  MoveL 1279 to (-195.45, 422.54, -1.48) mm, rotated rx 180 ry 0 rz 13.5 deg; joints [-3.576, -31.782, 134.338, -181.987, 89.848, 89.481, 155.176]
  MoveL 1280 to (-195.21, 422.52, -1.48) mm, rotated rx -180 ry 0 rz 13.48 deg; joints [-3.576, -31.791, 134.342, -181.987, 89.843, 89.481, 155.202]
  MoveL 1281 to (-194.97, 422.52, -1.48) mm, rotated rx 180 ry 0 rz 13.45 deg; joints [-3.576, -31.8, 134.346, -181.987, 89.838, 89.481, 155.229]
  Set speed (38.1 mm/s)
  MoveL 1282 to (-194.97, 421.25, -1.48) mm, rotated rx 180 ry 0 rz 13.52 deg; joints [-3.576, -31.894, 134.387, -181.987, 89.785, 89.483, 155.164]
  MoveL 1283 to (-195.61, 421.25, -1.47) mm, rotated rx 180 ry 0 rz 13.59 deg; joints [-3.576, -31.872, 134.377, -181.987, 89.798, 89.482, 155.093]
  Set speed (25.4 mm/s)
  MoveL 1284 to (-195.61, 421.25, -3.84) mm, rotated rx -180 ry 0 rz 13.59 deg; joints [-3.707, -31.873, 134.372, -182.114, 89.79, 89.454, 155.093]
  MoveL 1285 to (-195.61, 421.89, -4.48) mm, rotated rx 180 ry 0 rz 13.55 deg; joints [-3.742, -31.826, 134.349, -182.149, 89.814, 89.446, 155.125]
  Set speed (38.1 mm/s)
  MoveL 1286 to (-194.97, 422.52, -4.48) mm, rotated rx 180 ry 0 rz 13.45 deg; joints [-3.742, -31.8, 134.338, -182.149, 89.829, 89.445, 155.229]
  Set speed (76.2 mm/s)
  MoveL 1287 to (213.41, 422.52, -4.48) mm, rotated rx -180 ry 0 rz -38.12 deg; joints [-4.097, -49.127, 150.45, -182.187, 60.817, 89.337, 179]
  MoveL 1288 to (213.89, 422.53, -4.48) mm, rotated rx 180 ry 0 rz -38.17 deg; joints [-4.098, -49.152, 150.476, -182.187, 60.765, 89.336, 179]
  MoveL 1289 to (214.13, 422.55, -4.47) mm, rotated rx -180 ry 0 rz -38.19 deg; joints [-4.098, -49.161, 150.488, -182.187, 60.743, 89.336, 179]
  MoveL 1290 to (214.37, 422.59, -4.48) mm, rotated rx 180 ry 0 rz -38.22 deg; joints [-4.099, -49.169, 150.501, -182.187, 60.725, 89.336, 179]
  MoveL 1291 to (214.61, 422.65, -4.48) mm, rotated rx -180 ry 0 rz -38.24 deg; joints [-4.099, -49.173, 150.512, -182.187, 60.709, 89.335, 179]
  MoveL 1292 to (214.85, 422.74, -4.48) mm, rotated rx -180 ry 0 rz -38.26 deg; joints [-4.1, -49.175, 150.524, -182.187, 60.698, 89.334, 179]
  MoveL 1293 to (215.09, 422.84, -4.48) mm, rotated rx -180 ry 0 rz -38.28 deg; joints [-4.1, -49.174, 150.536, -182.187, 60.69, 89.334, 179]
  MoveL 1294 to (215.34, 422.97, -4.48) mm, rotated rx -180 ry 0 rz -38.3 deg; joints [-4.101, -49.17, 150.547, -182.187, 60.687, 89.333, 179]
  MoveL 1295 to (215.58, 423.13, -4.48) mm, rotated rx -180 ry 0 rz -38.32 deg; joints [-4.101, -49.161, 150.557, -182.186, 60.688, 89.332, 179]
  MoveL 1296 to (215.82, 423.33, -4.48) mm, rotated rx -180 ry 0 rz -38.33 deg; joints [-4.102, -49.148, 150.568, -182.186, 60.696, 89.33, 179]
  MoveL 1297 to (215.96, 423.46, -4.48) mm, rotated rx -180 ry 0 rz -38.34 deg; joints [-4.102, -49.138, 150.573, -182.186, 60.705, 89.33, 179]
  MoveL 1298 to (216.09, 423.6, -4.48) mm, rotated rx 180 ry 0 rz -38.35 deg; joints [-4.102, -49.127, 150.578, -182.186, 60.715, 89.329, 179]
  MoveL 1299 to (216.2, 423.73, -4.48) mm, rotated rx 180 ry 0 rz -38.35 deg; joints [-4.103, -49.115, 150.582, -182.186, 60.726, 89.328, 179]
  MoveL 1300 to (216.3, 423.87, -4.47) mm, rotated rx -180 ry 0 rz -38.36 deg; joints [-4.103, -49.102, 150.586, -182.186, 60.739, 89.327, 179]
  MoveL 1301 to (216.39, 424.01, -4.48) mm, rotated rx -180 ry 0 rz -38.36 deg; joints [-4.103, -49.089, 150.589, -182.185, 60.753, 89.326, 179]
  MoveL 1302 to (216.47, 424.15, -4.48) mm, rotated rx -180 ry 0 rz -38.36 deg; joints [-4.104, -49.075, 150.592, -182.185, 60.768, 89.326, 179]
  MoveL 1303 to (216.6, 424.39, -4.48) mm, rotated rx -180 ry 0 rz -38.36 deg; joints [-4.104, -49.049, 150.595, -182.185, 60.797, 89.324, 179]
  MoveL 1304 to (216.69, 424.63, -4.48) mm, rotated rx -180 ry 0 rz -38.36 deg; joints [-4.104, -49.023, 150.597, -182.185, 60.828, 89.323, 179]
  MoveL 1305 to (216.77, 424.87, -4.48) mm, rotated rx 180 ry 0 rz -38.35 deg; joints [-4.105, -48.995, 150.598, -182.185, 60.862, 89.322, 179]
  MoveL 1306 to (216.82, 425.11, -4.48) mm, rotated rx -180 ry 0 rz -38.34 deg; joints [-4.105, -48.966, 150.597, -182.184, 60.898, 89.32, 179]
  MoveL 1307 to (216.86, 425.35, -4.48) mm, rotated rx -180 ry 0 rz -38.33 deg; joints [-4.105, -48.936, 150.596, -182.184, 60.936, 89.319, 179]
  MoveL 1308 to (216.88, 425.59, -4.48) mm, rotated rx -180 ry 0 rz -38.32 deg; joints [-4.105, -48.905, 150.594, -182.184, 60.976, 89.318, 179]
  MoveL 1309 to (216.88, 426.08, -4.48) mm, rotated rx 180 ry 0 rz -38.3 deg; joints [-4.106, -48.841, 150.587, -182.183, 61.06, 89.315, 179]
  MoveL 1310 to (216.88, 426.56, -4.48) mm, rotated rx -180 ry 0 rz -38.27 deg; joints [-4.106, -48.777, 150.58, -182.183, 61.143, 89.313, 179]
  MoveL 1311 to (216.86, 426.8, -4.47) mm, rotated rx 180 ry 0 rz -38.26 deg; joints [-4.106, -48.744, 150.576, -182.182, 61.187, 89.312, 179]
  MoveL 1312 to (216.82, 427.04, -4.48) mm, rotated rx -180 ry 0 rz -38.24 deg; joints [-4.107, -48.71, 150.571, -182.182, 61.232, 89.311, 179]
  MoveL 1313 to (216.76, 427.29, -4.47) mm, rotated rx 180 ry 0 rz -38.22 deg; joints [-4.107, -48.675, 150.564, -182.182, 61.28, 89.31, 179]
  MoveL 1314 to (216.68, 427.53, -4.48) mm, rotated rx -180 ry 0 rz -38.2 deg; joints [-4.107, -48.639, 150.557, -182.182, 61.33, 89.308, 179]
  MoveL 1315 to (216.58, 427.77, -4.48) mm, rotated rx -180 ry 0 rz -38.17 deg; joints [-4.107, -48.602, 150.548, -182.182, 61.382, 89.307, 179]
  MoveL 1316 to (216.46, 428.01, -4.48) mm, rotated rx -180 ry 0 rz -38.15 deg; joints [-4.107, -48.564, 150.538, -182.181, 61.437, 89.306, 179]
  MoveL 1317 to (216.3, 428.26, -4.47) mm, rotated rx 180 ry 0 rz -38.12 deg; joints [-4.107, -48.523, 150.526, -182.181, 61.496, 89.305, 179]
  MoveL 1318 to (216.2, 428.39, -4.47) mm, rotated rx 180 ry 0 rz -38.1 deg; joints [-4.107, -48.5, 150.519, -182.181, 61.529, 89.305, 179]
  MoveL 1319 to (216.09, 428.53, -4.48) mm, rotated rx -180 ry 0 rz -38.08 deg; joints [-4.107, -48.476, 150.511, -182.181, 61.564, 89.304, 179]
  MoveL 1320 to (215.96, 428.66, -4.47) mm, rotated rx 180 ry 0 rz -38.06 deg; joints [-4.106, -48.452, 150.502, -182.181, 61.601, 89.304, 179]
  MoveL 1321 to (215.82, 428.8, -4.48) mm, rotated rx -180 ry 0 rz -38.04 deg; joints [-4.106, -48.427, 150.492, -182.181, 61.639, 89.303, 179]
  MoveL 1322 to (215.58, 428.99, -4.47) mm, rotated rx 180 ry 0 rz -38 deg; joints [-4.106, -48.389, 150.477, -182.18, 61.697, 89.303, 179]
  MoveL 1323 to (215.34, 429.15, -4.48) mm, rotated rx -180 ry 0 rz -37.97 deg; joints [-4.106, -48.355, 150.461, -182.18, 61.75, 89.302, 179]
  MoveL 1324 to (215.09, 429.28, -4.48) mm, rotated rx -180 ry 0 rz -37.93 deg; joints [-4.105, -48.326, 150.447, -182.18, 61.797, 89.302, 179]
  MoveL 1325 to (214.85, 429.39, -4.48) mm, rotated rx -180 ry 0 rz -37.9 deg; joints [-4.105, -48.299, 150.432, -182.18, 61.841, 89.301, 179]
  MoveL 1326 to (214.61, 429.47, -4.48) mm, rotated rx 180 ry 0 rz -37.87 deg; joints [-4.105, -48.276, 150.418, -182.18, 61.88, 89.301, 179]
  MoveL 1327 to (214.37, 429.53, -4.47) mm, rotated rx 180 ry 0 rz -37.84 deg; joints [-4.104, -48.255, 150.404, -182.18, 61.916, 89.301, 179]
  MoveL 1328 to (214.13, 429.58, -4.48) mm, rotated rx -180 ry 0 rz -37.82 deg; joints [-4.104, -48.237, 150.39, -182.18, 61.948, 89.301, 179]
  MoveL 1329 to (213.89, 429.6, -4.48) mm, rotated rx -180 ry 0 rz -37.79 deg; joints [-4.104, -48.222, 150.377, -182.18, 61.977, 89.302, 179]
  MoveL 1330 to (213.41, 429.6, -4.47) mm, rotated rx 180 ry 0 rz -37.74 deg; joints [-4.103, -48.196, 150.351, -182.18, 62.029, 89.302, 179]
  MoveL 1331 to (-194.97, 429.6, -4.48) mm, rotated rx 180 ry 0 rz 13.09 deg; joints [-3.743, -31.276, 134.105, -182.15, 90.119, 89.434, 155.59]
  MoveL 1332 to (-195.21, 429.6, -4.48) mm, rotated rx 180 ry 0 rz 13.12 deg; joints [-3.743, -31.268, 134.101, -182.15, 90.124, 89.434, 155.563]
  MoveL 1333 to (-195.45, 429.58, -4.47) mm, rotated rx -180 ry 0 rz 13.14 deg; joints [-3.743, -31.261, 134.098, -182.15, 90.128, 89.434, 155.535]
  MoveL 1334 to (-195.69, 429.55, -4.47) mm, rotated rx 180 ry 0 rz 13.17 deg; joints [-3.743, -31.256, 134.096, -182.15, 90.131, 89.434, 155.507]
  MoveL 1335 to (-195.93, 429.49, -4.48) mm, rotated rx 180 ry 0 rz 13.2 deg; joints [-3.743, -31.252, 134.094, -182.15, 90.133, 89.434, 155.477]
  MoveL 1336 to (-196.18, 429.42, -4.48) mm, rotated rx 180 ry 0 rz 13.23 deg; joints [-3.743, -31.249, 134.093, -182.15, 90.134, 89.434, 155.447]
  MoveL 1337 to (-196.42, 429.32, -4.48) mm, rotated rx 180 ry 0 rz 13.26 deg; joints [-3.743, -31.248, 134.092, -182.15, 90.135, 89.434, 155.415]
  MoveL 1338 to (-196.6, 429.23, -4.48) mm, rotated rx -180 ry 0 rz 13.29 deg; joints [-3.743, -31.249, 134.092, -182.15, 90.134, 89.434, 155.391]
  MoveL 1339 to (-196.78, 429.13, -4.48) mm, rotated rx 180 ry 0 rz 13.31 deg; joints [-3.743, -31.25, 134.093, -182.15, 90.133, 89.434, 155.366]
  MoveL 1340 to (-196.95, 429.01, -4.48) mm, rotated rx 180 ry 0 rz 13.34 deg; joints [-3.743, -31.253, 134.094, -182.15, 90.132, 89.434, 155.34]
  MoveL 1341 to (-197.13, 428.87, -4.48) mm, rotated rx 180 ry 0 rz 13.37 deg; joints [-3.743, -31.257, 134.096, -182.15, 90.13, 89.434, 155.313]
  MoveL 1342 to (-197.37, 428.65, -4.48) mm, rotated rx 180 ry 0 rz 13.4 deg; joints [-3.743, -31.265, 134.1, -182.15, 90.125, 89.434, 155.277]
  MoveL 1343 to (-197.56, 428.44, -4.48) mm, rotated rx -180 ry 0 rz 13.43 deg; joints [-3.743, -31.274, 134.104, -182.15, 90.12, 89.434, 155.245]
  MoveL 1344 to (-197.72, 428.22, -4.48) mm, rotated rx 180 ry 0 rz 13.46 deg; joints [-3.742, -31.285, 134.109, -182.15, 90.114, 89.434, 155.217]
  MoveL 1345 to (-197.85, 428.01, -4.47) mm, rotated rx 180 ry 0 rz 13.49 deg; joints [-3.742, -31.296, 134.114, -182.15, 90.108, 89.435, 155.191]
  MoveL 1346 to (-197.98, 427.77, -4.48) mm, rotated rx 180 ry 0 rz 13.51 deg; joints [-3.742, -31.31, 134.12, -182.15, 90.101, 89.435, 155.165]
  MoveL 1347 to (-198.08, 427.53, -4.48) mm, rotated rx 180 ry 0 rz 13.54 deg; joints [-3.742, -31.324, 134.126, -182.15, 90.093, 89.435, 155.141]
  MoveL 1348 to (-198.16, 427.29, -4.48) mm, rotated rx 180 ry 0 rz 13.56 deg; joints [-3.742, -31.339, 134.133, -182.15, 90.085, 89.435, 155.12]
  MoveL 1349 to (-198.21, 427.04, -4.48) mm, rotated rx 180 ry 0 rz 13.58 deg; joints [-3.742, -31.355, 134.14, -182.149, 90.076, 89.436, 155.102]
  MoveL 1350 to (-198.25, 426.8, -4.48) mm, rotated rx 180 ry 0 rz 13.59 deg; joints [-3.742, -31.372, 134.148, -182.149, 90.067, 89.436, 155.085]
  MoveL 1351 to (-198.27, 426.56, -4.48) mm, rotated rx -180 ry 0 rz 13.61 deg; joints [-3.742, -31.389, 134.155, -182.149, 90.057, 89.437, 155.071]
  MoveL 1352 to (-198.27, 426.08, -4.48) mm, rotated rx -180 ry 0 rz 13.63 deg; joints [-3.742, -31.424, 134.171, -182.149, 90.038, 89.437, 155.045]
  MoveL 1353 to (-198.27, 425.59, -4.48) mm, rotated rx 180 ry 0 rz 13.66 deg; joints [-3.742, -31.46, 134.187, -182.149, 90.018, 89.438, 155.021]
  MoveL 1354 to (-198.25, 425.35, -4.48) mm, rotated rx -180 ry 0 rz 13.67 deg; joints [-3.742, -31.478, 134.195, -182.149, 90.008, 89.438, 155.01]
  MoveL 1355 to (-198.22, 425.11, -4.48) mm, rotated rx -180 ry 0 rz 13.68 deg; joints [-3.742, -31.497, 134.204, -182.149, 89.997, 89.439, 155.002]
  MoveL 1356 to (-198.16, 424.87, -4.48) mm, rotated rx 180 ry 0 rz 13.68 deg; joints [-3.742, -31.517, 134.213, -182.149, 89.986, 89.439, 154.995]
  MoveL 1357 to (-198.09, 424.63, -4.48) mm, rotated rx -180 ry 0 rz 13.69 deg; joints [-3.742, -31.538, 134.222, -182.149, 89.975, 89.44, 154.991]
  MoveL 1358 to (-197.99, 424.39, -4.48) mm, rotated rx 180 ry 0 rz 13.69 deg; joints [-3.742, -31.559, 134.231, -182.149, 89.963, 89.44, 154.989]
  MoveL 1359 to (-197.87, 424.15, -4.47) mm, rotated rx 180 ry 0 rz 13.69 deg; joints [-3.742, -31.581, 134.241, -182.149, 89.951, 89.441, 154.991]
  MoveL 1360 to (-197.73, 423.93, -4.48) mm, rotated rx -180 ry 0 rz 13.69 deg; joints [-3.742, -31.602, 134.25, -182.149, 89.939, 89.441, 154.994]
  MoveL 1361 to (-197.57, 423.71, -4.48) mm, rotated rx 180 ry 0 rz 13.68 deg; joints [-3.742, -31.623, 134.26, -182.149, 89.927, 89.441, 155.001]
  MoveL 1362 to (-197.38, 423.49, -4.48) mm, rotated rx 180 ry 0 rz 13.67 deg; joints [-3.742, -31.646, 134.27, -182.149, 89.914, 89.442, 155.011]
  MoveL 1363 to (-197.14, 423.27, -4.48) mm, rotated rx -180 ry 0 rz 13.65 deg; joints [-3.742, -31.671, 134.281, -182.149, 89.901, 89.442, 155.026]
  MoveL 1364 to (-196.96, 423.13, -4.47) mm, rotated rx 180 ry 0 rz 13.64 deg; joints [-3.742, -31.687, 134.288, -182.149, 89.892, 89.443, 155.038]
  MoveL 1365 to (-196.78, 423, -4.47) mm, rotated rx 180 ry 0 rz 13.63 deg; joints [-3.742, -31.703, 134.295, -182.149, 89.883, 89.443, 155.052]
  MoveL 1366 to (-196.6, 422.9, -4.47) mm, rotated rx 180 ry 0 rz 13.61 deg; joints [-3.742, -31.717, 134.301, -182.149, 89.875, 89.443, 155.067]
  MoveL 1367 to (-196.42, 422.81, -4.48) mm, rotated rx -180 ry 0 rz 13.6 deg; joints [-3.742, -31.73, 134.307, -182.149, 89.868, 89.444, 155.083]
  MoveL 1368 to (-196.18, 422.71, -4.48) mm, rotated rx -180 ry 0 rz 13.58 deg; joints [-3.742, -31.745, 134.314, -182.149, 89.859, 89.444, 155.104]
  MoveL 1369 to (-195.93, 422.63, -4.48) mm, rotated rx 180 ry 0 rz 13.55 deg; joints [-3.742, -31.759, 134.32, -182.149, 89.852, 89.444, 155.127]
  MoveL 1370 to (-195.69, 422.58, -4.47) mm, rotated rx 180 ry 0 rz 13.53 deg; joints [-3.742, -31.771, 134.325, -182.149, 89.845, 89.445, 155.151]
  MoveL 1371 to (-195.45, 422.54, -4.48) mm, rotated rx 180 ry 0 rz 13.5 deg; joints [-3.742, -31.782, 134.33, -182.149, 89.839, 89.445, 155.176]
  MoveL 1372 to (-195.21, 422.52, -4.48) mm, rotated rx 180 ry 0 rz 13.48 deg; joints [-3.742, -31.792, 134.335, -182.149, 89.833, 89.445, 155.202]
  MoveL 1373 to (-194.97, 422.52, -4.48) mm, rotated rx 180 ry 0 rz 13.45 deg; joints [-3.742, -31.8, 134.338, -182.149, 89.829, 89.445, 155.229]
  Set speed (38.1 mm/s)
  MoveL 1374 to (-194.97, 421.25, -4.48) mm, rotated rx -180 ry 0 rz 13.52 deg; joints [-3.742, -31.894, 134.38, -182.149, 89.776, 89.447, 155.164]
  MoveL 1375 to (-195.61, 421.25, -4.48) mm, rotated rx -180 ry 0 rz 13.59 deg; joints [-3.742, -31.873, 134.37, -182.149, 89.788, 89.447, 155.093]
  Set speed (25.4 mm/s)
  MoveL 1376 to (-195.61, 421.25, -6.84) mm, rotated rx 180 ry 0 rz 13.59 deg; joints [-3.872, -31.873, 134.364, -182.276, 89.78, 89.419, 155.093]
  MoveL 1377 to (-195.61, 421.89, -7.47) mm, rotated rx 180 ry 0 rz 13.55 deg; joints [-3.907, -31.826, 134.341, -182.311, 89.804, 89.41, 155.125]
  Set speed (38.1 mm/s)
  MoveL 1378 to (-194.97, 422.52, -7.48) mm, rotated rx 180 ry 0 rz 13.45 deg; joints [-3.907, -31.801, 134.33, -182.311, 89.818, 89.41, 155.229]
  Set speed (76.2 mm/s)
  MoveL 1379 to (213.41, 422.52, -7.47) mm, rotated rx 180 ry 0 rz -38.12 deg; joints [-4.291, -49.127, 150.441, -182.356, 60.805, 89.294, 179]
  MoveL 1380 to (213.89, 422.53, -7.48) mm, rotated rx -180 ry 0 rz -38.17 deg; joints [-4.291, -49.152, 150.466, -182.356, 60.754, 89.293, 179]
  MoveL 1381 to (214.13, 422.55, -7.48) mm, rotated rx -180 ry 0 rz -38.19 deg; joints [-4.292, -49.162, 150.479, -182.356, 60.732, 89.293, 179]
  MoveL 1382 to (214.37, 422.59, -7.48) mm, rotated rx 180 ry 0 rz -38.22 deg; joints [-4.292, -49.169, 150.491, -182.356, 60.713, 89.293, 179]
  MoveL 1383 to (214.61, 422.65, -7.48) mm, rotated rx -180 ry 0 rz -38.24 deg; joints [-4.293, -49.174, 150.503, -182.356, 60.698, 89.292, 179]
  MoveL 1384 to (214.85, 422.74, -7.47) mm, rotated rx 180 ry 0 rz -38.26 deg; joints [-4.293, -49.176, 150.515, -182.356, 60.686, 89.291, 179]
  MoveL 1385 to (215.09, 422.84, -7.47) mm, rotated rx 180 ry 0 rz -38.28 deg; joints [-4.294, -49.175, 150.526, -182.355, 60.678, 89.29, 179]
  MoveL 1386 to (215.34, 422.97, -7.48) mm, rotated rx -180 ry 0 rz -38.3 deg; joints [-4.294, -49.17, 150.537, -182.355, 60.675, 89.289, 179]
  MoveL 1387 to (215.58, 423.13, -7.48) mm, rotated rx -180 ry 0 rz -38.32 deg; joints [-4.295, -49.162, 150.548, -182.355, 60.677, 89.288, 179]
  MoveL 1388 to (215.82, 423.33, -7.47) mm, rotated rx 180 ry 0 rz -38.33 deg; joints [-4.296, -49.149, 150.558, -182.355, 60.685, 89.287, 179]
  MoveL 1389 to (215.96, 423.46, -7.48) mm, rotated rx -180 ry 0 rz -38.34 deg; joints [-4.296, -49.139, 150.564, -182.355, 60.693, 89.286, 179]
  MoveL 1390 to (216.09, 423.6, -7.48) mm, rotated rx -180 ry 0 rz -38.35 deg; joints [-4.296, -49.128, 150.569, -182.355, 60.703, 89.285, 179]
  MoveL 1391 to (216.2, 423.73, -7.48) mm, rotated rx 180 ry 0 rz -38.35 deg; joints [-4.297, -49.116, 150.573, -182.354, 60.714, 89.284, 179]
  MoveL 1392 to (216.3, 423.87, -7.48) mm, rotated rx -180 ry 0 rz -38.36 deg; joints [-4.297, -49.103, 150.577, -182.354, 60.727, 89.283, 179]
  MoveL 1393 to (216.39, 424.01, -7.48) mm, rotated rx 180 ry 0 rz -38.36 deg; joints [-4.297, -49.09, 150.58, -182.354, 60.741, 89.283, 179]
  MoveL 1394 to (216.47, 424.15, -7.48) mm, rotated rx -180 ry 0 rz -38.36 deg; joints [-4.298, -49.076, 150.582, -182.354, 60.756, 89.282, 179]
  MoveL 1395 to (216.6, 424.39, -7.48) mm, rotated rx -180 ry 0 rz -38.36 deg; joints [-4.298, -49.05, 150.585, -182.354, 60.785, 89.28, 179]
  MoveL 1396 to (216.69, 424.63, -7.48) mm, rotated rx 180 ry 0 rz -38.36 deg; joints [-4.298, -49.024, 150.587, -182.353, 60.817, 89.279, 179]
  MoveL 1397 to (216.77, 424.87, -7.47) mm, rotated rx -180 ry 0 rz -38.35 deg; joints [-4.299, -48.996, 150.588, -182.353, 60.85, 89.277, 179]
  MoveL 1398 to (216.82, 425.11, -7.47) mm, rotated rx -180 ry 0 rz -38.34 deg; joints [-4.299, -48.967, 150.588, -182.353, 60.886, 89.276, 179]
  MoveL 1399 to (216.86, 425.35, -7.48) mm, rotated rx -180 ry 0 rz -38.33 deg; joints [-4.299, -48.937, 150.587, -182.353, 60.924, 89.275, 179]
  MoveL 1400 to (216.88, 425.59, -7.47) mm, rotated rx 180 ry 0 rz -38.32 deg; joints [-4.3, -48.906, 150.584, -182.352, 60.964, 89.273, 179]
  MoveL 1401 to (216.88, 426.08, -7.48) mm, rotated rx -180 ry 0 rz -38.3 deg; joints [-4.3, -48.842, 150.578, -182.352, 61.048, 89.271, 179]
  MoveL 1402 to (216.88, 427.04, -7.47) mm, rotated rx 180 ry 0 rz -38.24 deg; joints [-4.301, -48.714, 150.564, -182.351, 61.214, 89.266, 179]
  MoveL 1403 to (216.86, 427.29, -7.48) mm, rotated rx -180 ry 0 rz -38.23 deg; joints [-4.301, -48.682, 150.56, -182.35, 61.257, 89.264, 179]
  MoveL 1404 to (216.83, 427.53, -7.48) mm, rotated rx -180 ry 0 rz -38.21 deg; joints [-4.301, -48.648, 150.555, -182.35, 61.302, 89.263, 179]
  MoveL 1405 to (216.78, 427.77, -7.48) mm, rotated rx -180 ry 0 rz -38.19 deg; joints [-4.301, -48.614, 150.549, -182.35, 61.349, 89.262, 179]
  MoveL 1406 to (216.71, 428.01, -7.47) mm, rotated rx 180 ry 0 rz -38.17 deg; joints [-4.301, -48.578, 150.542, -182.35, 61.398, 89.261, 179]
  MoveL 1407 to (216.63, 428.21, -7.48) mm, rotated rx -180 ry 0 rz -38.16 deg; joints [-4.301, -48.548, 150.535, -182.349, 61.441, 89.26, 179]
  MoveL 1408 to (216.54, 428.41, -7.48) mm, rotated rx 180 ry 0 rz -38.13 deg; joints [-4.301, -48.517, 150.527, -182.349, 61.484, 89.259, 179]
  MoveL 1409 to (216.43, 428.61, -7.48) mm, rotated rx 180 ry 0 rz -38.11 deg; joints [-4.301, -48.485, 150.518, -182.349, 61.53, 89.258, 179]
  MoveL 1410 to (216.3, 428.81, -7.48) mm, rotated rx -180 ry 0 rz -38.09 deg; joints [-4.301, -48.452, 150.509, -182.349, 61.578, 89.257, 179]
  MoveL 1411 to (216.16, 428.99, -7.48) mm, rotated rx -180 ry 0 rz -38.06 deg; joints [-4.301, -48.42, 150.498, -182.348, 61.624, 89.256, 179]
  MoveL 1412 to (215.99, 429.18, -7.48) mm, rotated rx -180 ry 0 rz -38.04 deg; joints [-4.301, -48.387, 150.487, -182.348, 61.673, 89.255, 179]
  MoveL 1413 to (215.78, 429.38, -7.48) mm, rotated rx -180 ry 0 rz -38 deg; joints [-4.301, -48.35, 150.473, -182.348, 61.729, 89.255, 179]
  MoveL 1414 to (215.57, 429.55, -7.48) mm, rotated rx -180 ry 0 rz -37.97 deg; joints [-4.301, -48.317, 150.459, -182.348, 61.78, 89.254, 179]
  MoveL 1415 to (215.39, 429.67, -7.48) mm, rotated rx -180 ry 0 rz -37.94 deg; joints [-4.3, -48.291, 150.447, -182.348, 61.82, 89.254, 179]
  MoveL 1416 to (215.21, 429.78, -7.48) mm, rotated rx -180 ry 0 rz -37.92 deg; joints [-4.3, -48.268, 150.436, -182.348, 61.857, 89.253, 179]
  MoveL 1417 to (215.02, 429.87, -7.47) mm, rotated rx 180 ry 0 rz -37.9 deg; joints [-4.3, -48.246, 150.425, -182.348, 61.892, 89.253, 179]
  MoveL 1418 to (214.84, 429.94, -7.48) mm, rotated rx -180 ry 0 rz -37.87 deg; joints [-4.3, -48.227, 150.414, -182.348, 61.924, 89.253, 179]
  MoveL 1419 to (214.61, 430.02, -7.48) mm, rotated rx 180 ry 0 rz -37.84 deg; joints [-4.299, -48.204, 150.4, -182.347, 61.962, 89.253, 179]
  MoveL 1420 to (214.37, 430.08, -7.47) mm, rotated rx 180 ry 0 rz -37.81 deg; joints [-4.299, -48.184, 150.387, -182.347, 61.997, 89.253, 179]
  MoveL 1421 to (214.13, 430.13, -7.47) mm, rotated rx 180 ry 0 rz -37.79 deg; joints [-4.298, -48.166, 150.373, -182.347, 62.029, 89.253, 179]
  MoveL 1422 to (213.89, 430.15, -7.48) mm, rotated rx -180 ry 0 rz -37.76 deg; joints [-4.298, -48.151, 150.36, -182.347, 62.058, 89.253, 179]
  MoveL 1423 to (213.41, 430.15, -7.48) mm, rotated rx -180 ry 0 rz -37.71 deg; joints [-4.297, -48.125, 150.334, -182.347, 62.11, 89.254, 179]
  MoveL 1424 to (-194.49, 430.15, -7.48) mm, rotated rx -180 ry 0 rz 13.01 deg; joints [-3.908, -31.252, 134.086, -182.311, 90.123, 89.397, 155.671]
  MoveL 1425 to (-195.36, 430.14, -7.48) mm, rotated rx -180 ry 0 rz 13.11 deg; joints [-3.908, -31.223, 134.073, -182.311, 90.138, 89.397, 155.573]
  MoveL 1426 to (-195.58, 430.12, -7.48) mm, rotated rx 180 ry 0 rz 13.13 deg; joints [-3.908, -31.218, 134.07, -182.311, 90.141, 89.396, 155.548]
  MoveL 1427 to (-195.8, 430.08, -7.48) mm, rotated rx 180 ry 0 rz 13.16 deg; joints [-3.908, -31.214, 134.068, -182.311, 90.144, 89.396, 155.522]
  MoveL 1428 to (-196.02, 430.02, -7.47) mm, rotated rx 180 ry 0 rz 13.18 deg; joints [-3.908, -31.211, 134.067, -182.311, 90.146, 89.396, 155.495]
  MoveL 1429 to (-196.24, 429.94, -7.47) mm, rotated rx 180 ry 0 rz 13.21 deg; joints [-3.908, -31.209, 134.066, -182.311, 90.147, 89.396, 155.467]
  MoveL 1430 to (-196.42, 429.87, -7.48) mm, rotated rx 180 ry 0 rz 13.24 deg; joints [-3.908, -31.208, 134.066, -182.311, 90.147, 89.396, 155.443]
  MoveL 1431 to (-196.56, 429.79, -7.48) mm, rotated rx 180 ry 0 rz 13.26 deg; joints [-3.908, -31.209, 134.066, -182.311, 90.147, 89.396, 155.423]
  MoveL 1432 to (-196.71, 429.71, -7.48) mm, rotated rx 180 ry 0 rz 13.28 deg; joints [-3.908, -31.21, 134.067, -182.311, 90.146, 89.396, 155.403]
  MoveL 1433 to (-196.86, 429.62, -7.48) mm, rotated rx 180 ry 0 rz 13.3 deg; joints [-3.908, -31.212, 134.068, -182.311, 90.145, 89.396, 155.382]
  MoveL 1434 to (-197.01, 429.52, -7.48) mm, rotated rx 180 ry 0 rz 13.32 deg; joints [-3.908, -31.214, 134.069, -182.311, 90.144, 89.396, 155.36]
  MoveL 1435 to (-197.15, 429.4, -7.48) mm, rotated rx 180 ry 0 rz 13.34 deg; joints [-3.908, -31.218, 134.07, -182.311, 90.141, 89.396, 155.338]
  MoveL 1436 to (-197.3, 429.27, -7.48) mm, rotated rx 180 ry 0 rz 13.36 deg; joints [-3.908, -31.223, 134.073, -182.311, 90.139, 89.396, 155.315]
  MoveL 1437 to (-197.46, 429.1, -7.48) mm, rotated rx 180 ry 0 rz 13.39 deg; joints [-3.908, -31.23, 134.076, -182.311, 90.135, 89.397, 155.29]
  MoveL 1438 to (-197.6, 428.94, -7.48) mm, rotated rx 180 ry 0 rz 13.41 deg; joints [-3.908, -31.237, 134.079, -182.311, 90.131, 89.397, 155.266]
  MoveL 1439 to (-197.76, 428.71, -7.48) mm, rotated rx 180 ry 0 rz 13.44 deg; joints [-3.908, -31.248, 134.084, -182.311, 90.125, 89.397, 155.236]
  MoveL 1440 to (-197.9, 428.47, -7.48) mm, rotated rx 180 ry 0 rz 13.47 deg; joints [-3.908, -31.261, 134.09, -182.311, 90.118, 89.397, 155.209]
  MoveL 1441 to (-198.01, 428.24, -7.47) mm, rotated rx -180 ry 0 rz 13.49 deg; joints [-3.908, -31.274, 134.096, -182.311, 90.111, 89.398, 155.185]
  MoveL 1442 to (-198.1, 428.01, -7.48) mm, rotated rx 180 ry 0 rz 13.52 deg; joints [-3.908, -31.288, 134.102, -182.311, 90.103, 89.398, 155.163]
  MoveL 1443 to (-198.17, 427.77, -7.47) mm, rotated rx -180 ry 0 rz 13.54 deg; joints [-3.908, -31.304, 134.109, -182.311, 90.094, 89.398, 155.143]
  MoveL 1444 to (-198.23, 427.53, -7.47) mm, rotated rx -180 ry 0 rz 13.55 deg; joints [-3.908, -31.32, 134.116, -182.311, 90.086, 89.399, 155.125]
  MoveL 1445 to (-198.26, 427.29, -7.48) mm, rotated rx -180 ry 0 rz 13.57 deg; joints [-3.908, -31.336, 134.124, -182.311, 90.076, 89.399, 155.109]
  MoveL 1446 to (-198.27, 427.04, -7.48) mm, rotated rx 180 ry 0 rz 13.58 deg; joints [-3.908, -31.354, 134.131, -182.311, 90.067, 89.399, 155.095]
  MoveL 1447 to (-198.27, 426.08, -7.48) mm, rotated rx -180 ry 0 rz 13.63 deg; joints [-3.908, -31.425, 134.163, -182.311, 90.027, 89.401, 155.045]
  MoveL 1448 to (-198.27, 425.59, -7.48) mm, rotated rx 180 ry 0 rz 13.66 deg; joints [-3.908, -31.461, 134.179, -182.311, 90.008, 89.402, 155.021]
  MoveL 1449 to (-198.25, 425.35, -7.48) mm, rotated rx -180 ry 0 rz 13.67 deg; joints [-3.908, -31.479, 134.187, -182.311, 89.997, 89.402, 155.01]
  MoveL 1450 to (-198.22, 425.11, -7.48) mm, rotated rx 180 ry 0 rz 13.68 deg; joints [-3.908, -31.498, 134.196, -182.311, 89.987, 89.403, 155.002]
  MoveL 1451 to (-198.16, 424.87, -7.47) mm, rotated rx 180 ry 0 rz 13.68 deg; joints [-3.908, -31.518, 134.205, -182.311, 89.976, 89.403, 154.995]
  MoveL 1452 to (-198.09, 424.63, -7.48) mm, rotated rx -180 ry 0 rz 13.69 deg; joints [-3.908, -31.538, 134.214, -182.311, 89.965, 89.404, 154.991]
  MoveL 1453 to (-197.99, 424.39, -7.48) mm, rotated rx -180 ry 0 rz 13.69 deg; joints [-3.908, -31.56, 134.223, -182.311, 89.953, 89.404, 154.989]
  MoveL 1454 to (-197.87, 424.15, -7.47) mm, rotated rx 180 ry 0 rz 13.69 deg; joints [-3.908, -31.582, 134.233, -182.311, 89.941, 89.405, 154.991]
  MoveL 1455 to (-197.73, 423.93, -7.47) mm, rotated rx 180 ry 0 rz 13.69 deg; joints [-3.908, -31.602, 134.242, -182.311, 89.929, 89.405, 154.994]
  MoveL 1456 to (-197.57, 423.71, -7.47) mm, rotated rx 180 ry 0 rz 13.68 deg; joints [-3.908, -31.624, 134.252, -182.311, 89.917, 89.406, 155.001]
  MoveL 1457 to (-197.38, 423.49, -7.48) mm, rotated rx -180 ry 0 rz 13.67 deg; joints [-3.908, -31.647, 134.262, -182.311, 89.904, 89.406, 155.011]
  MoveL 1458 to (-197.14, 423.27, -7.47) mm, rotated rx 180 ry 0 rz 13.65 deg; joints [-3.908, -31.671, 134.273, -182.311, 89.891, 89.407, 155.026]
  MoveL 1459 to (-196.96, 423.13, -7.48) mm, rotated rx -180 ry 0 rz 13.64 deg; joints [-3.908, -31.688, 134.28, -182.311, 89.881, 89.407, 155.038]
  MoveL 1460 to (-196.78, 423, -7.47) mm, rotated rx 180 ry 0 rz 13.63 deg; joints [-3.908, -31.703, 134.287, -182.311, 89.873, 89.407, 155.052]
  MoveL 1461 to (-196.6, 422.9, -7.47) mm, rotated rx 180 ry 0 rz 13.61 deg; joints [-3.908, -31.717, 134.293, -182.311, 89.865, 89.408, 155.067]
  MoveL 1462 to (-196.42, 422.81, -7.48) mm, rotated rx 180 ry 0 rz 13.6 deg; joints [-3.908, -31.73, 134.299, -182.311, 89.858, 89.408, 155.083]
  MoveL 1463 to (-196.18, 422.71, -7.48) mm, rotated rx -180 ry 0 rz 13.58 deg; joints [-3.908, -31.746, 134.306, -182.311, 89.849, 89.408, 155.104]
  MoveL 1464 to (-195.93, 422.63, -7.48) mm, rotated rx -180 ry 0 rz 13.55 deg; joints [-3.908, -31.76, 134.312, -182.311, 89.842, 89.409, 155.127]
  MoveL 1465 to (-195.69, 422.58, -7.48) mm, rotated rx -180 ry 0 rz 13.53 deg; joints [-3.908, -31.772, 134.317, -182.311, 89.835, 89.409, 155.151]
  MoveL 1466 to (-195.45, 422.54, -7.48) mm, rotated rx 180 ry 0 rz 13.5 deg; joints [-3.908, -31.783, 134.322, -182.311, 89.829, 89.409, 155.176]
  MoveL 1467 to (-195.21, 422.52, -7.47) mm, rotated rx -180 ry 0 rz 13.48 deg; joints [-3.908, -31.793, 134.327, -182.311, 89.823, 89.409, 155.202]
  MoveL 1468 to (-194.97, 422.52, -7.48) mm, rotated rx 180 ry 0 rz 13.45 deg; joints [-3.907, -31.801, 134.33, -182.311, 89.818, 89.41, 155.229]
  Set speed (38.1 mm/s)
  MoveL 1469 to (-194.97, 421.25, -7.48) mm, rotated rx -180 ry 0 rz 13.52 deg; joints [-3.907, -31.895, 134.372, -182.31, 89.766, 89.412, 155.164]
  MoveL 1470 to (-195.61, 421.25, -7.47) mm, rotated rx 180 ry 0 rz 13.59 deg; joints [-3.907, -31.873, 134.362, -182.31, 89.778, 89.411, 155.093]
  Set speed (25.4 mm/s)
  MoveL 1471 to (-195.61, 421.25, -9.84) mm, rotated rx 180 ry 0 rz 13.59 deg; joints [-4.038, -31.874, 134.355, -182.438, 89.77, 89.383, 155.093]
  MoveL 1472 to (-195.61, 421.89, -10.48) mm, rotated rx -180 ry 0 rz 13.55 deg; joints [-4.073, -31.827, 134.333, -182.472, 89.794, 89.375, 155.125]
  Set speed (38.1 mm/s)
  MoveL 1473 to (-194.97, 422.52, -10.48) mm, rotated rx 180 ry 0 rz 13.45 deg; joints [-4.073, -31.802, 134.322, -182.472, 89.808, 89.374, 155.229]
  Set speed (76.2 mm/s)
  MoveL 1474 to (213.41, 422.52, -10.48) mm, rotated rx -180 ry 0 rz -38.12 deg; joints [-4.484, -49.128, 150.431, -182.524, 60.792, 89.251, 179]
  MoveL 1475 to (213.89, 422.53, -10.48) mm, rotated rx -180 ry 0 rz -38.17 deg; joints [-4.485, -49.153, 150.456, -182.524, 60.741, 89.251, 179]
  MoveL 1476 to (214.13, 422.55, -10.48) mm, rotated rx 180 ry 0 rz -38.19 deg; joints [-4.485, -49.163, 150.469, -182.524, 60.719, 89.25, 179]
  MoveL 1477 to (214.37, 422.59, -10.47) mm, rotated rx 180 ry 0 rz -38.22 deg; joints [-4.486, -49.17, 150.481, -182.524, 60.7, 89.25, 179]
  MoveL 1478 to (214.61, 422.65, -10.48) mm, rotated rx -180 ry 0 rz -38.24 deg; joints [-4.486, -49.175, 150.493, -182.524, 60.685, 89.249, 179]
  MoveL 1479 to (214.85, 422.74, -10.48) mm, rotated rx -180 ry 0 rz -38.26 deg; joints [-4.487, -49.177, 150.505, -182.524, 60.673, 89.248, 179]
  MoveL 1480 to (215.09, 422.84, -10.48) mm, rotated rx 180 ry 0 rz -38.28 deg; joints [-4.488, -49.176, 150.516, -182.524, 60.666, 89.247, 179]
  MoveL 1481 to (215.34, 422.97, -10.48) mm, rotated rx -180 ry 0 rz -38.3 deg; joints [-4.488, -49.171, 150.527, -182.524, 60.662, 89.246, 179]
  MoveL 1482 to (215.58, 423.13, -10.48) mm, rotated rx 180 ry 0 rz -38.32 deg; joints [-4.489, -49.163, 150.538, -182.524, 60.664, 89.245, 179]
  MoveL 1483 to (215.82, 423.33, -10.48) mm, rotated rx -180 ry 0 rz -38.33 deg; joints [-4.489, -49.15, 150.548, -182.524, 60.672, 89.244, 179]
  MoveL 1484 to (215.96, 423.46, -10.48) mm, rotated rx -180 ry 0 rz -38.34 deg; joints [-4.49, -49.14, 150.554, -182.523, 60.68, 89.243, 179]
  MoveL 1485 to (216.09, 423.6, -10.48) mm, rotated rx 180 ry 0 rz -38.35 deg; joints [-4.49, -49.128, 150.559, -182.523, 60.69, 89.242, 179]
  MoveL 1486 to (216.2, 423.73, -10.48) mm, rotated rx -180 ry 0 rz -38.35 deg; joints [-4.491, -49.117, 150.563, -182.523, 60.702, 89.241, 179]
  MoveL 1487 to (216.3, 423.87, -10.48) mm, rotated rx -180 ry 0 rz -38.36 deg; joints [-4.491, -49.104, 150.566, -182.523, 60.714, 89.24, 179]
  MoveL 1488 to (216.39, 424.01, -10.47) mm, rotated rx 180 ry 0 rz -38.36 deg; joints [-4.491, -49.091, 150.569, -182.523, 60.728, 89.239, 179]
  MoveL 1489 to (216.47, 424.15, -10.48) mm, rotated rx -180 ry 0 rz -38.36 deg; joints [-4.491, -49.077, 150.572, -182.523, 60.744, 89.238, 179]
  MoveL 1490 to (216.69, 424.27, -10.47) mm, rotated rx 180 ry 0 rz -38.38 deg; joints [-4.492, -49.072, 150.582, -182.522, 60.741, 89.237, 179]
  MoveL 1491 to (219.83, 424.27, -10.48) mm, rotated rx -180 ry 0 rz -38.71 deg; joints [-4.498, -49.236, 150.748, -182.523, 60.408, 89.233, 179]
  MoveL 1492 to (220.05, 424.15, -10.47) mm, rotated rx 180 ry 0 rz -38.74 deg; joints [-4.498, -49.264, 150.761, -182.523, 60.363, 89.233, 179]
  MoveL 1493 to (220.05, 53.41, -10.47) mm, rotated rx -180 ry 0 rz -47.68 deg; joints [-4.3, -87.184, 146.455, -190.693, 9.341, 98.376, 179]
  MoveL 1494 to (219.83, 53.17, -10.47) mm, rotated rx 180 ry 0 rz -47.72 deg; joints [-4.299, -87.185, 146.415, -190.774, 9.257, 98.458, 179]
  MoveL 1495 to (-199.12, 53.17, -10.47) mm, rotated rx 180 ry 0 rz 63.73 deg; joints [-4.039, -53.792, 140.61, -182.536, 74.12, 90.068, 104.952]
  MoveL 1496 to (-199.7, 53.18, -10.48) mm, rotated rx -180 ry 0 rz 63.77 deg; joints [-4.039, -53.744, 140.603, -182.536, 74.162, 90.066, 104.91]
  MoveL 1497 to (-199.9, 53.41, -10.48) mm, rotated rx -180 ry 0 rz 63.72 deg; joints [-4.039, -53.723, 140.6, -182.535, 74.18, 90.065, 104.959]
  MoveL 1498 to (-199.9, 424.15, -10.48) mm, rotated rx 180 ry 0 rz 13.91 deg; joints [-4.074, -31.512, 134.193, -182.473, 89.969, 89.367, 154.766]
  MoveL 1499 to (-199.7, 424.27, -10.48) mm, rotated rx 180 ry 0 rz 13.89 deg; joints [-4.074, -31.51, 134.192, -182.473, 89.97, 89.367, 154.794]
  MoveL 1500 to (-198.11, 424.27, -10.48) mm, rotated rx -180 ry 0 rz 13.71 deg; joints [-4.074, -31.565, 134.217, -182.473, 89.939, 89.368, 154.97]
  MoveL 1501 to (-197.87, 424.15, -10.48) mm, rotated rx 180 ry 0 rz 13.69 deg; joints [-4.074, -31.582, 134.225, -182.473, 89.93, 89.369, 154.991]
  MoveL 1502 to (-197.73, 423.93, -10.48) mm, rotated rx -180 ry 0 rz 13.69 deg; joints [-4.074, -31.603, 134.234, -182.473, 89.918, 89.369, 154.994]
  MoveL 1503 to (-197.57, 423.71, -10.48) mm, rotated rx 180 ry 0 rz 13.68 deg; joints [-4.074, -31.625, 134.243, -182.473, 89.906, 89.37, 155.001]
  MoveL 1504 to (-197.38, 423.49, -10.48) mm, rotated rx 180 ry 0 rz 13.67 deg; joints [-4.073, -31.648, 134.254, -182.472, 89.893, 89.37, 155.011]
  MoveL 1505 to (-197.14, 423.27, -10.48) mm, rotated rx 180 ry 0 rz 13.65 deg; joints [-4.073, -31.672, 134.264, -182.472, 89.88, 89.371, 155.026]
  MoveL 1506 to (-196.96, 423.13, -10.48) mm, rotated rx -180 ry 0 rz 13.64 deg; joints [-4.073, -31.689, 134.272, -182.472, 89.871, 89.371, 155.038]
  MoveL 1507 to (-196.78, 423, -10.48) mm, rotated rx 180 ry 0 rz 13.63 deg; joints [-4.073, -31.704, 134.279, -182.472, 89.862, 89.372, 155.052]
  MoveL 1508 to (-196.6, 422.9, -10.48) mm, rotated rx 180 ry 0 rz 13.61 deg; joints [-4.073, -31.718, 134.285, -182.472, 89.854, 89.372, 155.067]
  MoveL 1509 to (-196.42, 422.81, -10.47) mm, rotated rx -180 ry 0 rz 13.6 deg; joints [-4.073, -31.731, 134.29, -182.472, 89.847, 89.372, 155.083]
  MoveL 1510 to (-196.18, 422.71, -10.48) mm, rotated rx -180 ry 0 rz 13.58 deg; joints [-4.073, -31.747, 134.297, -182.472, 89.838, 89.373, 155.104]
  MoveL 1511 to (-195.93, 422.63, -10.48) mm, rotated rx -180 ry 0 rz 13.55 deg; joints [-4.073, -31.761, 134.303, -182.472, 89.831, 89.373, 155.127]
  MoveL 1512 to (-195.69, 422.58, -10.48) mm, rotated rx -180 ry 0 rz 13.53 deg; joints [-4.073, -31.773, 134.309, -182.472, 89.824, 89.373, 155.151]
  MoveL 1513 to (-195.45, 422.54, -10.48) mm, rotated rx 180 ry 0 rz 13.5 deg; joints [-4.073, -31.784, 134.314, -182.472, 89.818, 89.374, 155.176]
  MoveL 1514 to (-195.21, 422.52, -10.48) mm, rotated rx 180 ry 0 rz 13.48 deg; joints [-4.073, -31.794, 134.318, -182.472, 89.812, 89.374, 155.202]
  MoveL 1515 to (-194.97, 422.52, -10.48) mm, rotated rx 180 ry 0 rz 13.45 deg; joints [-4.073, -31.802, 134.322, -182.472, 89.808, 89.374, 155.229]
  Set speed (38.1 mm/s)
  MoveL 1516 to (-194.97, 421.25, -10.48) mm, rotated rx 180 ry 0 rz 13.52 deg; joints [-4.073, -31.896, 134.363, -182.472, 89.755, 89.376, 155.164]
  MoveL 1517 to (-195.61, 421.25, -10.48) mm, rotated rx 180 ry 0 rz 13.59 deg; joints [-4.073, -31.874, 134.354, -182.472, 89.767, 89.376, 155.093]
  Set speed (25.4 mm/s)
  MoveL 1518 to (-195.61, 421.25, -12.84) mm, rotated rx 180 ry 0 rz 13.59 deg; joints [-4.204, -31.875, 134.346, -182.6, 89.758, 89.348, 155.093]
  MoveL 1519 to (-195.61, 421.89, -13.47) mm, rotated rx 180 ry 0 rz 13.55 deg; joints [-4.239, -31.828, 134.324, -182.634, 89.782, 89.339, 155.125]
  Set speed (38.1 mm/s)
  MoveL 1520 to (-194.97, 422.52, -13.48) mm, rotated rx 180 ry 0 rz 13.45 deg; joints [-4.239, -31.803, 134.313, -182.634, 89.796, 89.339, 155.229]
  Set speed (76.2 mm/s)
  MoveL 1521 to (213.41, 422.52, -13.48) mm, rotated rx -180 ry 0 rz -38.12 deg; joints [-4.677, -49.129, 150.42, -182.693, 60.779, 89.208, 179]
  MoveL 1522 to (213.89, 422.53, -13.47) mm, rotated rx -180 ry 0 rz -38.17 deg; joints [-4.678, -49.154, 150.445, -182.693, 60.728, 89.208, 179]
  MoveL 1523 to (214.13, 422.55, -13.48) mm, rotated rx -180 ry 0 rz -38.19 deg; joints [-4.679, -49.164, 150.458, -182.693, 60.706, 89.207, 179]
  MoveL 1524 to (214.37, 422.59, -13.48) mm, rotated rx -180 ry 0 rz -38.22 deg; joints [-4.679, -49.171, 150.47, -182.693, 60.687, 89.207, 179]
  MoveL 1525 to (214.61, 422.65, -13.48) mm, rotated rx -180 ry 0 rz -38.24 deg; joints [-4.68, -49.176, 150.482, -182.693, 60.672, 89.206, 179]
  MoveL 1526 to (214.85, 422.74, -13.48) mm, rotated rx -180 ry 0 rz -38.26 deg; joints [-4.681, -49.178, 150.494, -182.693, 60.66, 89.205, 179]
  MoveL 1527 to (215.09, 422.84, -13.48) mm, rotated rx -180 ry 0 rz -38.28 deg; joints [-4.681, -49.176, 150.505, -182.693, 60.652, 89.204, 179]
  MoveL 1528 to (215.34, 422.97, -13.48) mm, rotated rx -180 ry 0 rz -38.3 deg; joints [-4.682, -49.172, 150.516, -182.693, 60.649, 89.203, 179]
  MoveL 1529 to (215.58, 423.13, -13.47) mm, rotated rx 180 ry 0 rz -38.32 deg; joints [-4.682, -49.164, 150.527, -182.693, 60.651, 89.202, 179]
  MoveL 1530 to (215.82, 423.33, -13.47) mm, rotated rx 180 ry 0 rz -38.33 deg; joints [-4.683, -49.151, 150.537, -182.692, 60.659, 89.2, 179]
  MoveL 1531 to (215.96, 423.46, -13.48) mm, rotated rx -180 ry 0 rz -38.34 deg; joints [-4.684, -49.14, 150.543, -182.692, 60.667, 89.199, 179]
  MoveL 1532 to (216.09, 423.6, -13.47) mm, rotated rx -180 ry 0 rz -38.35 deg; joints [-4.684, -49.129, 150.548, -182.692, 60.677, 89.198, 179]
  MoveL 1533 to (216.2, 423.73, -13.48) mm, rotated rx -180 ry 0 rz -38.35 deg; joints [-4.684, -49.117, 150.552, -182.692, 60.688, 89.197, 179]
  MoveL 1534 to (216.3, 423.87, -13.48) mm, rotated rx -180 ry 0 rz -38.36 deg; joints [-4.685, -49.105, 150.556, -182.692, 60.701, 89.196, 179]
  MoveL 1535 to (216.39, 424.01, -13.48) mm, rotated rx -180 ry 0 rz -38.36 deg; joints [-4.685, -49.091, 150.559, -182.691, 60.715, 89.195, 179]
  MoveL 1536 to (216.47, 424.15, -13.47) mm, rotated rx 180 ry 0 rz -38.36 deg; joints [-4.685, -49.077, 150.561, -182.691, 60.73, 89.194, 179]
  MoveL 1537 to (216.69, 424.27, -13.48) mm, rotated rx -180 ry 0 rz -38.38 deg; joints [-4.686, -49.073, 150.571, -182.691, 60.728, 89.193, 179]
  MoveL 1538 to (219.83, 424.27, -13.48) mm, rotated rx 180 ry 0 rz -38.71 deg; joints [-4.692, -49.237, 150.737, -182.691, 60.395, 89.189, 179]
  MoveL 1539 to (220.05, 424.15, -13.47) mm, rotated rx 180 ry 0 rz -38.74 deg; joints [-4.693, -49.265, 150.75, -182.691, 60.35, 89.19, 179]
  MoveL 1540 to (220.05, 53.41, -13.47) mm, rotated rx -180 ry 0 rz -47.68 deg; joints [-4.484, -87.175, 146.444, -191.411, 9.358, 98.944, 179]
  MoveL 1541 to (219.83, 53.17, -13.48) mm, rotated rx 180 ry 0 rz -47.72 deg; joints [-4.482, -87.176, 146.405, -191.497, 9.274, 99.031, 179]
  MoveL 1542 to (-197.29, 53.18, -13.48) mm, rotated rx -180 ry 0 rz 63.6 deg; joints [-4.204, -53.942, 140.62, -182.705, 73.981, 90.084, 105.084]
  MoveL 1543 to (-197.94, 53.17, -13.47) mm, rotated rx 180 ry 0 rz 63.64 deg; joints [-4.204, -53.888, 140.613, -182.704, 74.028, 90.082, 105.037]
  MoveL 1544 to (-198.16, 53.41, -13.48) mm, rotated rx -180 ry 0 rz 63.6 deg; joints [-4.204, -53.865, 140.61, -182.704, 74.048, 90.081, 105.084]
  MoveL 1545 to (-198.16, 424.15, -13.48) mm, rotated rx 180 ry 0 rz 13.72 deg; joints [-4.239, -31.573, 134.211, -182.634, 89.924, 89.333, 154.958]
  MoveL 1546 to (-198.01, 424.27, -13.48) mm, rotated rx 180 ry 0 rz 13.7 deg; joints [-4.239, -31.569, 134.209, -182.634, 89.926, 89.333, 154.981]
  MoveL 1547 to (-197.87, 424.15, -13.47) mm, rotated rx 180 ry 0 rz 13.69 deg; joints [-4.239, -31.583, 134.215, -182.634, 89.918, 89.333, 154.991]
  MoveL 1548 to (-197.73, 423.93, -13.48) mm, rotated rx -180 ry 0 rz 13.69 deg; joints [-4.239, -31.604, 134.225, -182.634, 89.907, 89.334, 154.994]
  MoveL 1549 to (-197.57, 423.71, -13.47) mm, rotated rx -180 ry 0 rz 13.68 deg; joints [-4.239, -31.626, 134.234, -182.634, 89.895, 89.334, 155.001]
  MoveL 1550 to (-197.38, 423.49, -13.48) mm, rotated rx -180 ry 0 rz 13.67 deg; joints [-4.239, -31.649, 134.244, -182.634, 89.882, 89.335, 155.011]
  MoveL 1551 to (-197.22, 423.33, -13.48) mm, rotated rx -180 ry 0 rz 13.66 deg; joints [-4.239, -31.666, 134.252, -182.634, 89.873, 89.335, 155.021]
  MoveL 1552 to (-197.14, 423.27, -13.48) mm, rotated rx 180 ry 0 rz 13.65 deg; joints [-4.239, -31.673, 134.255, -182.634, 89.868, 89.335, 155.026]
  MoveL 1553 to (-196.96, 423.13, -13.48) mm, rotated rx 180 ry 0 rz 13.64 deg; joints [-4.239, -31.69, 134.263, -182.634, 89.859, 89.336, 155.038]
  MoveL 1554 to (-196.78, 423, -13.48) mm, rotated rx 180 ry 0 rz 13.63 deg; joints [-4.239, -31.705, 134.269, -182.634, 89.851, 89.336, 155.052]
  MoveL 1555 to (-196.6, 422.9, -13.48) mm, rotated rx -180 ry 0 rz 13.61 deg; joints [-4.239, -31.719, 134.276, -182.634, 89.843, 89.336, 155.067]
  MoveL 1556 to (-196.42, 422.81, -13.47) mm, rotated rx 180 ry 0 rz 13.6 deg; joints [-4.239, -31.732, 134.281, -182.634, 89.836, 89.337, 155.083]
  MoveL 1557 to (-196.18, 422.71, -13.47) mm, rotated rx -180 ry 0 rz 13.58 deg; joints [-4.239, -31.747, 134.288, -182.634, 89.827, 89.337, 155.104]
  MoveL 1558 to (-195.93, 422.63, -13.48) mm, rotated rx -180 ry 0 rz 13.55 deg; joints [-4.239, -31.761, 134.294, -182.634, 89.819, 89.338, 155.127]
  MoveL 1559 to (-195.69, 422.58, -13.47) mm, rotated rx 180 ry 0 rz 13.53 deg; joints [-4.239, -31.774, 134.3, -182.634, 89.812, 89.338, 155.151]
  MoveL 1560 to (-195.45, 422.54, -13.47) mm, rotated rx 180 ry 0 rz 13.5 deg; joints [-4.239, -31.785, 134.305, -182.634, 89.806, 89.338, 155.176]
  MoveL 1561 to (-195.21, 422.52, -13.47) mm, rotated rx 180 ry 0 rz 13.48 deg; joints [-4.239, -31.794, 134.309, -182.634, 89.801, 89.338, 155.202]
  MoveL 1562 to (-194.97, 422.52, -13.47) mm, rotated rx 180 ry 0 rz 13.45 deg; joints [-4.239, -31.803, 134.313, -182.634, 89.796, 89.339, 155.229]
  Set speed (38.1 mm/s)
  MoveL 1563 to (-194.97, 421.25, -13.48) mm, rotated rx 180 ry 0 rz 13.52 deg; joints [-4.239, -31.897, 134.354, -182.634, 89.744, 89.341, 155.164]
  MoveL 1564 to (-195.61, 421.25, -13.47) mm, rotated rx 180 ry 0 rz 13.59 deg; joints [-4.239, -31.875, 134.344, -182.634, 89.756, 89.341, 155.093]
  Set speed (25.4 mm/s)
  MoveL 1565 to (-195.61, 421.25, -15.84) mm, rotated rx 180 ry 0 rz 13.59 deg; joints [-4.369, -31.876, 134.337, -182.761, 89.746, 89.313, 155.093]
  MoveL 1566 to (-195.61, 421.89, -16.48) mm, rotated rx 180 ry 0 rz 13.55 deg; joints [-4.405, -31.829, 134.314, -182.795, 89.77, 89.304, 155.125]
  Set speed (38.1 mm/s)
  MoveL 1567 to (-194.97, 422.52, -16.48) mm, rotated rx 180 ry 0 rz 13.45 deg; joints [-4.405, -31.804, 134.303, -182.795, 89.784, 89.303, 155.229]
  Set speed (76.2 mm/s)
  MoveL 1568 to (213.41, 422.52, -16.47) mm, rotated rx 180 ry 0 rz -38.12 deg; joints [-4.871, -49.13, 150.408, -182.862, 60.765, 89.166, 179]
  MoveL 1569 to (213.89, 422.53, -16.48) mm, rotated rx -180 ry 0 rz -38.17 deg; joints [-4.872, -49.155, 150.434, -182.862, 60.714, 89.165, 179]
  MoveL 1570 to (214.13, 422.55, -16.48) mm, rotated rx -180 ry 0 rz -38.19 deg; joints [-4.872, -49.165, 150.446, -182.862, 60.692, 89.165, 179]
  MoveL 1571 to (214.37, 422.59, -16.48) mm, rotated rx -180 ry 0 rz -38.22 deg; joints [-4.873, -49.172, 150.459, -182.862, 60.673, 89.164, 179]
  MoveL 1572 to (214.61, 422.65, -16.48) mm, rotated rx 180 ry 0 rz -38.24 deg; joints [-4.873, -49.176, 150.47, -182.862, 60.658, 89.163, 179]
  MoveL 1573 to (214.85, 422.74, -16.47) mm, rotated rx 180 ry 0 rz -38.26 deg; joints [-4.874, -49.178, 150.482, -182.862, 60.646, 89.162, 179]
  MoveL 1574 to (215.09, 422.84, -16.47) mm, rotated rx 180 ry 0 rz -38.28 deg; joints [-4.875, -49.177, 150.494, -182.862, 60.638, 89.161, 179]
  MoveL 1575 to (215.34, 422.97, -16.47) mm, rotated rx -180 ry 0 rz -38.3 deg; joints [-4.875, -49.173, 150.505, -182.861, 60.635, 89.16, 179]
  MoveL 1576 to (215.58, 423.13, -16.48) mm, rotated rx -180 ry 0 rz -38.32 deg; joints [-4.876, -49.165, 150.515, -182.861, 60.637, 89.159, 179]
  MoveL 1577 to (215.82, 423.33, -16.48) mm, rotated rx -180 ry 0 rz -38.33 deg; joints [-4.877, -49.152, 150.526, -182.861, 60.644, 89.157, 179]
  MoveL 1578 to (215.96, 423.46, -16.48) mm, rotated rx -180 ry 0 rz -38.34 deg; joints [-4.877, -49.141, 150.531, -182.861, 60.653, 89.156, 179]
  MoveL 1579 to (216.09, 423.6, -16.47) mm, rotated rx -180 ry 0 rz -38.35 deg; joints [-4.878, -49.13, 150.536, -182.861, 60.663, 89.155, 179]
  MoveL 1580 to (216.2, 423.73, -16.48) mm, rotated rx -180 ry 0 rz -38.35 deg; joints [-4.878, -49.118, 150.54, -182.86, 60.674, 89.154, 179]
  MoveL 1581 to (216.3, 423.87, -16.47) mm, rotated rx -180 ry 0 rz -38.36 deg; joints [-4.878, -49.106, 150.544, -182.86, 60.687, 89.153, 179]
  MoveL 1582 to (216.39, 424.01, -16.48) mm, rotated rx 180 ry 0 rz -38.36 deg; joints [-4.879, -49.092, 150.547, -182.86, 60.701, 89.152, 179]
  MoveL 1583 to (216.47, 424.15, -16.47) mm, rotated rx -180 ry 0 rz -38.36 deg; joints [-4.879, -49.078, 150.55, -182.86, 60.716, 89.151, 179]
  MoveL 1584 to (216.69, 424.27, -16.48) mm, rotated rx -180 ry 0 rz -38.38 deg; joints [-4.88, -49.074, 150.56, -182.86, 60.713, 89.15, 179]
  MoveL 1585 to (219.83, 424.27, -16.47) mm, rotated rx -180 ry 0 rz -38.71 deg; joints [-4.887, -49.238, 150.725, -182.86, 60.38, 89.145, 179]
  MoveL 1586 to (220.05, 424.15, -16.47) mm, rotated rx -180 ry 0 rz -38.74 deg; joints [-4.887, -49.266, 150.739, -182.86, 60.335, 89.146, 179]
  MoveL 1587 to (220.05, 53.41, -16.47) mm, rotated rx -180 ry 0 rz -47.68 deg; joints [-4.667, -87.165, 146.433, -192.127, 9.376, 99.509, 179]
  MoveL 1588 to (219.83, 53.18, -16.47) mm, rotated rx -180 ry 0 rz -47.72 deg; joints [-4.666, -87.166, 146.394, -192.218, 9.293, 99.602, 179]
  MoveL 1589 to (-196.42, 53.17, -16.47) mm, rotated rx 180 ry 0 rz 63.53 deg; joints [-4.368, -54.012, 140.619, -182.873, 73.911, 90.098, 105.148]
  MoveL 1590 to (-196.42, 53.41, -16.47) mm, rotated rx 180 ry 0 rz 63.47 deg; joints [-4.368, -54.006, 140.618, -182.873, 73.916, 90.097, 105.211]
  MoveL 1591 to (-196.42, 422.66, -16.47) mm, rotated rx 180 ry 0 rz 13.61 deg; joints [-4.405, -31.744, 134.276, -182.796, 89.817, 89.302, 155.075]
  MoveL 1592 to (-196.42, 422.81, -16.48) mm, rotated rx 180 ry 0 rz 13.6 deg; joints [-4.405, -31.733, 134.272, -182.796, 89.823, 89.301, 155.083]
  MoveL 1593 to (-196.18, 422.71, -16.48) mm, rotated rx 180 ry 0 rz 13.58 deg; joints [-4.405, -31.748, 134.279, -182.796, 89.815, 89.302, 155.104]
  MoveL 1594 to (-195.93, 422.63, -16.47) mm, rotated rx 180 ry 0 rz 13.55 deg; joints [-4.405, -31.762, 134.285, -182.796, 89.807, 89.302, 155.127]
  MoveL 1595 to (-195.69, 422.58, -16.48) mm, rotated rx -180 ry 0 rz 13.53 deg; joints [-4.405, -31.775, 134.29, -182.796, 89.8, 89.303, 155.151]
  MoveL 1596 to (-195.45, 422.54, -16.47) mm, rotated rx 180 ry 0 rz 13.5 deg; joints [-4.405, -31.786, 134.295, -182.795, 89.794, 89.303, 155.176]
  MoveL 1597 to (-195.21, 422.52, -16.48) mm, rotated rx 180 ry 0 rz 13.48 deg; joints [-4.405, -31.795, 134.299, -182.795, 89.789, 89.303, 155.202]
  MoveL 1598 to (-194.97, 422.52, -16.48) mm, rotated rx 180 ry 0 rz 13.45 deg; joints [-4.405, -31.804, 134.303, -182.795, 89.784, 89.303, 155.229]
  MoveL 1599 to (-164.9, 422.52, -17.53) mm, rotated rx 180 ry 0 rz 10 deg; joints [-4.461, -32.767, 134.717, -182.851, 89.235, 89.318, 158.68]
  MoveL 1600 to (213.41, 422.52, -17.53) mm, rotated rx -180 ry 0 rz -38.12 deg; joints [-4.938, -49.13, 150.404, -182.921, 60.76, 89.151, 179]
  MoveL 1601 to (213.89, 422.53, -17.52) mm, rotated rx 180 ry 0 rz -38.17 deg; joints [-4.939, -49.155, 150.43, -182.921, 60.708, 89.15, 179]
  MoveL 1602 to (214.13, 422.55, -17.53) mm, rotated rx -180 ry 0 rz -38.19 deg; joints [-4.94, -49.165, 150.442, -182.921, 60.686, 89.15, 179]
  MoveL 1603 to (214.37, 422.59, -17.53) mm, rotated rx -180 ry 0 rz -38.22 deg; joints [-4.94, -49.172, 150.454, -182.921, 60.668, 89.149, 179]
  MoveL 1604 to (214.61, 422.65, -17.53) mm, rotated rx -180 ry 0 rz -38.24 deg; joints [-4.941, -49.177, 150.466, -182.921, 60.652, 89.148, 179]
  MoveL 1605 to (214.85, 422.74, -17.53) mm, rotated rx -180 ry 0 rz -38.26 deg; joints [-4.942, -49.179, 150.478, -182.921, 60.641, 89.147, 179]
  MoveL 1606 to (215.09, 422.84, -17.53) mm, rotated rx -180 ry 0 rz -38.28 deg; joints [-4.942, -49.178, 150.489, -182.921, 60.633, 89.146, 179]
  MoveL 1607 to (215.34, 422.97, -17.52) mm, rotated rx 180 ry 0 rz -38.3 deg; joints [-4.943, -49.173, 150.5, -182.921, 60.63, 89.145, 179]
  MoveL 1608 to (215.58, 423.13, -17.53) mm, rotated rx -180 ry 0 rz -38.32 deg; joints [-4.944, -49.165, 150.511, -182.92, 60.631, 89.144, 179]
  MoveL 1609 to (215.82, 423.33, -17.53) mm, rotated rx -180 ry 0 rz -38.33 deg; joints [-4.944, -49.152, 150.521, -182.92, 60.639, 89.142, 179]
  MoveL 1610 to (215.96, 423.46, -17.53) mm, rotated rx -180 ry 0 rz -38.34 deg; joints [-4.945, -49.142, 150.527, -182.92, 60.647, 89.141, 179]
  MoveL 1611 to (216.09, 423.6, -17.53) mm, rotated rx -180 ry 0 rz -38.35 deg; joints [-4.945, -49.13, 150.532, -182.92, 60.657, 89.14, 179]
  MoveL 1612 to (216.2, 423.73, -17.53) mm, rotated rx -180 ry 0 rz -38.35 deg; joints [-4.946, -49.119, 150.536, -182.919, 60.669, 89.139, 179]
  MoveL 1613 to (216.3, 423.87, -17.52) mm, rotated rx -180 ry 0 rz -38.36 deg; joints [-4.946, -49.106, 150.54, -182.919, 60.681, 89.138, 179]
  MoveL 1614 to (216.39, 424.01, -17.53) mm, rotated rx 180 ry 0 rz -38.36 deg; joints [-4.946, -49.093, 150.543, -182.919, 60.696, 89.137, 179]
  MoveL 1615 to (216.47, 424.15, -17.53) mm, rotated rx -180 ry 0 rz -38.36 deg; joints [-4.947, -49.079, 150.545, -182.919, 60.711, 89.136, 179]
  MoveL 1616 to (216.69, 424.27, -17.52) mm, rotated rx -180 ry 0 rz -38.38 deg; joints [-4.947, -49.074, 150.555, -182.919, 60.708, 89.135, 179]
  MoveL 1617 to (219.83, 424.27, -17.53) mm, rotated rx -180 ry 0 rz -38.71 deg; joints [-4.955, -49.238, 150.721, -182.919, 60.375, 89.13, 179]
  MoveL 1618 to (220.05, 424.15, -17.53) mm, rotated rx 180 ry 0 rz -38.74 deg; joints [-4.955, -49.266, 150.735, -182.919, 60.33, 89.131, 179]
  MoveL 1619 to (220.05, 53.41, -17.52) mm, rotated rx -180 ry 0 rz -47.68 deg; joints [-4.731, -87.161, 146.429, -192.376, 9.382, 99.706, 179]
  MoveL 1620 to (219.83, 53.18, -17.52) mm, rotated rx -180 ry 0 rz -47.72 deg; joints [-4.73, -87.162, 146.39, -192.469, 9.299, 99.801, 179]
  MoveL 1621 to (-195.15, 53.17, -17.53) mm, rotated rx -180 ry 0 rz 63.44 deg; joints [-4.426, -54.115, 140.628, -182.932, 73.817, 90.106, 105.242]
  MoveL 1622 to (-195.65, 53.17, -17.52) mm, rotated rx 180 ry 0 rz 63.47 deg; joints [-4.426, -54.074, 140.623, -182.932, 73.853, 90.104, 105.205]
  MoveL 1623 to (-195.81, 53.41, -17.53) mm, rotated rx 180 ry 0 rz 63.42 deg; joints [-4.426, -54.055, 140.621, -182.932, 73.869, 90.103, 105.256]
  MoveL 1624 to (-195.81, 422.38, -17.53) mm, rotated rx 180 ry 0 rz 13.55 deg; joints [-4.463, -31.786, 134.291, -182.852, 89.79, 89.29, 155.128]
  MoveL 1625 to (-195.65, 422.57, -17.53) mm, rotated rx 180 ry 0 rz 13.52 deg; joints [-4.463, -31.777, 134.288, -182.852, 89.794, 89.29, 155.156]
  MoveL 1626 to (-195.48, 422.55, -17.53) mm, rotated rx 180 ry 0 rz 13.51 deg; joints [-4.463, -31.785, 134.291, -182.852, 89.79, 89.29, 155.173]
  MoveL 1627 to (-195.32, 422.53, -17.53) mm, rotated rx -180 ry 0 rz 13.49 deg; joints [-4.463, -31.791, 134.294, -182.852, 89.786, 89.291, 155.191]
  MoveL 1628 to (-195.15, 422.52, -17.53) mm, rotated rx -180 ry 0 rz 13.47 deg; joints [-4.463, -31.798, 134.297, -182.852, 89.783, 89.291, 155.209]
  MoveL 1629 to (-194.97, 422.52, -17.52) mm, rotated rx 180 ry 0 rz 13.45 deg; joints [-4.463, -31.804, 134.299, -182.852, 89.779, 89.291, 155.229]
  MoveL 1630 to (-164.9, 422.52, -17.53) mm, rotated rx 180 ry 0 rz 10 deg; joints [-4.461, -32.767, 134.717, -182.851, 89.235, 89.318, 158.68]
  Set speed (38.1 mm/s)
  MoveL 1631 to (-164.28, 421.77, -17.53) mm, rotated rx 180 ry 0 rz 9.96 deg; joints [-4.461, -32.843, 134.75, -182.851, 89.192, 89.321, 158.719]
  MoveL 1632 to (-164.81, 418.84, -17.53) mm, rotated rx -180 ry 0 rz 10.16 deg; joints [-4.46, -33.051, 134.838, -182.85, 89.072, 89.327, 158.52]
  MoveL 1633 to (-164.93, 418.21, -16.89) mm, rotated rx -180 ry 0 rz 10.2 deg; joints [-4.425, -33.095, 134.859, -182.816, 89.049, 89.335, 158.477]
  Set speed (100.0 mm/s)
  MoveL 1634 to (-164.93, 418.21, 24.52) mm, rotated rx -180 ry 0 rz 10.2 deg; joints [-2.136, -33.087, 134.943, -180.583, 89.155, 89.801, 158.477]
  MoveL 1635 to (-164.87, 434.05, 24.52) mm, rotated rx 180 ry 0 rz 9.48 deg; joints [-2.138, -31.879, 134.422, -180.584, 89.842, 89.793, 159.202]
  MoveL 1636 to (-164.87, 434.05, -6.52) mm, rotated rx -180 ry 0 rz 9.48 deg; joints [-3.854, -31.885, 134.37, -182.259, 89.775, 89.423, 159.202]
  Set speed (25.4 mm/s)
  MoveL 1637 to (-164.87, 434.05, -9.84) mm, rotated rx -180 ry 0 rz 9.48 deg; joints [-4.038, -31.886, 134.361, -182.438, 89.763, 89.384, 159.202]
  MoveL 1638 to (-164.72, 433.43, -10.47) mm, rotated rx 180 ry 0 rz 9.49 deg; joints [-4.073, -31.938, 134.382, -182.472, 89.732, 89.377, 159.191]
  Set speed (38.1 mm/s)
  MoveL 1639 to (-164.28, 431.48, -10.48) mm, rotated rx 180 ry 0 rz 9.52 deg; joints [-4.073, -32.099, 134.452, -182.472, 89.641, 89.381, 159.156]
  MoveL 1640 to (-164.9, 430.7, -10.48) mm, rotated rx -180 ry 0 rz 9.63 deg; joints [-4.073, -32.14, 134.47, -182.472, 89.618, 89.382, 159.05]
  Set speed (76.2 mm/s)
  MoveL 1641 to (-194.97, 430.7, -10.47) mm, rotated rx -180 ry 0 rz 13.03 deg; joints [-4.074, -31.196, 134.052, -182.473, 90.143, 89.359, 155.645]
  MoveL 1642 to (-202.2, 430.7, -10.48) mm, rotated rx 180 ry 0 rz 13.83 deg; joints [-4.075, -30.95, 133.94, -182.474, 90.278, 89.353, 154.851]
  MoveL 1643 to (-203.17, 430.7, -10.48) mm, rotated rx -180 ry 0 rz 13.93 deg; joints [-4.075, -30.917, 133.925, -182.474, 90.296, 89.353, 154.746]
  MoveL 1644 to (-203.41, 430.69, -10.47) mm, rotated rx 180 ry 0 rz 13.96 deg; joints [-4.075, -30.91, 133.922, -182.474, 90.3, 89.353, 154.719]
  MoveL 1645 to (-203.65, 430.65, -10.47) mm, rotated rx 180 ry 0 rz 13.99 deg; joints [-4.075, -30.904, 133.919, -182.474, 90.303, 89.352, 154.691]
  MoveL 1646 to (-203.89, 430.6, -10.48) mm, rotated rx 180 ry 0 rz 14.02 deg; joints [-4.075, -30.899, 133.917, -182.474, 90.305, 89.352, 154.662]
  MoveL 1647 to (-204.13, 430.52, -10.48) mm, rotated rx 180 ry 0 rz 14.05 deg; joints [-4.075, -30.896, 133.916, -182.474, 90.307, 89.352, 154.632]
  MoveL 1648 to (-204.42, 430.43, -10.48) mm, rotated rx 180 ry 0 rz 14.08 deg; joints [-4.075, -30.893, 133.915, -182.474, 90.309, 89.352, 154.595]
  MoveL 1649 to (-204.57, 430.37, -10.48) mm, rotated rx -180 ry 0 rz 14.1 deg; joints [-4.075, -30.892, 133.914, -182.474, 90.309, 89.352, 154.577]
  MoveL 1650 to (-204.72, 430.31, -10.47) mm, rotated rx 180 ry 0 rz 14.12 deg; joints [-4.075, -30.892, 133.914, -182.474, 90.309, 89.352, 154.557]
  MoveL 1651 to (-204.86, 430.23, -10.47) mm, rotated rx 180 ry 0 rz 14.14 deg; joints [-4.075, -30.892, 133.914, -182.474, 90.309, 89.352, 154.538]
  MoveL 1652 to (-205.01, 430.15, -10.48) mm, rotated rx 180 ry 0 rz 14.16 deg; joints [-4.075, -30.893, 133.915, -182.474, 90.309, 89.352, 154.517]
  MoveL 1653 to (-205.16, 430.05, -10.47) mm, rotated rx 180 ry 0 rz 14.18 deg; joints [-4.075, -30.895, 133.916, -182.474, 90.308, 89.352, 154.497]
  MoveL 1654 to (-205.3, 429.94, -10.48) mm, rotated rx 180 ry 0 rz 14.2 deg; joints [-4.075, -30.898, 133.917, -182.474, 90.306, 89.352, 154.475]
  MoveL 1655 to (-205.53, 429.75, -10.48) mm, rotated rx 180 ry 0 rz 14.24 deg; joints [-4.075, -30.904, 133.92, -182.474, 90.303, 89.352, 154.441]
  MoveL 1656 to (-205.75, 429.52, -10.47) mm, rotated rx 180 ry 0 rz 14.28 deg; joints [-4.075, -30.914, 133.924, -182.474, 90.298, 89.353, 154.404]
  MoveL 1657 to (-205.92, 429.3, -10.48) mm, rotated rx 180 ry 0 rz 14.3 deg; joints [-4.075, -30.923, 133.928, -182.474, 90.292, 89.353, 154.375]
  MoveL 1658 to (-206.06, 429.09, -10.48) mm, rotated rx -180 ry 0 rz 14.33 deg; joints [-4.075, -30.934, 133.933, -182.474, 90.287, 89.353, 154.348]
  MoveL 1659 to (-206.14, 428.95, -10.47) mm, rotated rx 180 ry 0 rz 14.35 deg; joints [-4.075, -30.941, 133.936, -182.474, 90.283, 89.353, 154.333]
  MoveL 1660 to (-206.21, 428.82, -10.48) mm, rotated rx 180 ry 0 rz 14.36 deg; joints [-4.075, -30.948, 133.94, -182.474, 90.279, 89.353, 154.319]
  MoveL 1661 to (-206.27, 428.69, -10.48) mm, rotated rx 180 ry 0 rz 14.37 deg; joints [-4.075, -30.956, 133.943, -182.474, 90.274, 89.354, 154.305]
  MoveL 1662 to (-206.32, 428.55, -10.47) mm, rotated rx 180 ry 0 rz 14.39 deg; joints [-4.075, -30.964, 133.947, -182.474, 90.27, 89.354, 154.292]
  MoveL 1663 to (-206.37, 428.42, -10.48) mm, rotated rx 180 ry 0 rz 14.4 deg; joints [-4.075, -30.972, 133.951, -182.474, 90.266, 89.354, 154.28]
  MoveL 1664 to (-206.41, 428.28, -10.48) mm, rotated rx 180 ry 0 rz 14.41 deg; joints [-4.075, -30.981, 133.954, -182.474, 90.261, 89.354, 154.268]
  MoveL 1665 to (-206.47, 428.01, -10.48) mm, rotated rx 180 ry 0 rz 14.43 deg; joints [-4.075, -30.998, 133.962, -182.474, 90.251, 89.355, 154.248]
  MoveL 1666 to (-206.5, 427.77, -10.48) mm, rotated rx -180 ry 0 rz 14.45 deg; joints [-4.075, -31.015, 133.97, -182.473, 90.242, 89.355, 154.231]
  MoveL 1667 to (-206.52, 427.53, -10.47) mm, rotated rx -180 ry 0 rz 14.46 deg; joints [-4.074, -31.032, 133.978, -182.473, 90.233, 89.355, 154.217]
  MoveL 1668 to (-206.52, 427.04, -10.48) mm, rotated rx -180 ry 0 rz 14.49 deg; joints [-4.074, -31.067, 133.994, -182.473, 90.214, 89.356, 154.191]
  MoveL 1669 to (-206.52, 50.21, -10.48) mm, rotated rx -180 ry 0 rz 65.02 deg; joints [-4.04, -53.239, 140.533, -182.531, 74.596, 90.046, 103.664]
  MoveL 1670 to (-206.51, 49.73, -10.48) mm, rotated rx 180 ry 0 rz 65.14 deg; joints [-4.04, -53.25, 140.535, -182.531, 74.587, 90.046, 103.539]
  MoveL 1671 to (-206.48, 49.48, -10.48) mm, rotated rx 180 ry 0 rz 65.2 deg; joints [-4.04, -53.257, 140.536, -182.531, 74.581, 90.046, 103.477]
  MoveL 1672 to (-206.43, 49.24, -10.48) mm, rotated rx 180 ry 0 rz 65.26 deg; joints [-4.04, -53.266, 140.537, -182.531, 74.573, 90.047, 103.417]
  MoveL 1673 to (-206.37, 49.02, -10.48) mm, rotated rx -180 ry 0 rz 65.32 deg; joints [-4.04, -53.276, 140.538, -182.531, 74.565, 90.047, 103.362]
  MoveL 1674 to (-206.28, 48.8, -10.48) mm, rotated rx -180 ry 0 rz 65.37 deg; joints [-4.04, -53.287, 140.54, -182.531, 74.555, 90.048, 103.309]
  MoveL 1675 to (-206.18, 48.57, -10.48) mm, rotated rx -180 ry 0 rz 65.42 deg; joints [-4.04, -53.3, 140.542, -182.532, 74.544, 90.048, 103.256]
  MoveL 1676 to (-206.06, 48.35, -10.48) mm, rotated rx -180 ry 0 rz 65.47 deg; joints [-4.04, -53.315, 140.544, -182.532, 74.531, 90.049, 103.205]
  MoveL 1677 to (-205.98, 48.22, -10.48) mm, rotated rx -180 ry 0 rz 65.5 deg; joints [-4.04, -53.324, 140.545, -182.532, 74.523, 90.049, 103.176]
  MoveL 1678 to (-205.88, 48.09, -10.48) mm, rotated rx 180 ry 0 rz 65.53 deg; joints [-4.04, -53.335, 140.547, -182.532, 74.514, 90.049, 103.148]
  MoveL 1679 to (-205.78, 47.96, -10.48) mm, rotated rx -180 ry 0 rz 65.56 deg; joints [-4.04, -53.346, 140.548, -182.532, 74.505, 90.05, 103.12]
  MoveL 1680 to (-205.66, 47.83, -10.48) mm, rotated rx -180 ry 0 rz 65.59 deg; joints [-4.04, -53.358, 140.55, -182.532, 74.494, 90.05, 103.092]
  MoveL 1681 to (-205.51, 47.67, -10.47) mm, rotated rx 180 ry 0 rz 65.62 deg; joints [-4.04, -53.374, 140.552, -182.532, 74.48, 90.051, 103.06]
  MoveL 1682 to (-205.35, 47.54, -10.47) mm, rotated rx 180 ry 0 rz 65.65 deg; joints [-4.04, -53.39, 140.554, -182.532, 74.467, 90.052, 103.034]
  MoveL 1683 to (-205.19, 47.42, -10.48) mm, rotated rx 180 ry 0 rz 65.67 deg; joints [-4.04, -53.406, 140.557, -182.532, 74.453, 90.052, 103.012]
  MoveL 1684 to (-205.03, 47.31, -10.48) mm, rotated rx -180 ry 0 rz 65.69 deg; joints [-4.04, -53.421, 140.559, -182.533, 74.44, 90.053, 102.993]
  MoveL 1685 to (-204.81, 47.18, -10.47) mm, rotated rx 180 ry 0 rz 65.71 deg; joints [-4.04, -53.442, 140.562, -182.533, 74.422, 90.054, 102.973]
  MoveL 1686 to (-204.58, 47.08, -10.48) mm, rotated rx 180 ry 0 rz 65.72 deg; joints [-4.04, -53.463, 140.565, -182.533, 74.404, 90.055, 102.958]
  MoveL 1687 to (-204.36, 46.99, -10.48) mm, rotated rx -180 ry 0 rz 65.73 deg; joints [-4.04, -53.484, 140.567, -182.533, 74.386, 90.055, 102.95]
  MoveL 1688 to (-204.13, 46.92, -10.48) mm, rotated rx -180 ry 0 rz 65.73 deg; joints [-4.04, -53.504, 140.57, -182.533, 74.369, 90.056, 102.946]
  MoveL 1689 to (-203.89, 46.87, -10.47) mm, rotated rx 180 ry 0 rz 65.73 deg; joints [-4.04, -53.525, 140.573, -182.534, 74.351, 90.057, 102.947]
  MoveL 1690 to (-203.65, 46.84, -10.48) mm, rotated rx 180 ry 0 rz 65.73 deg; joints [-4.04, -53.546, 140.576, -182.534, 74.333, 90.058, 102.953]
  MoveL 1691 to (-203.41, 46.83, -10.48) mm, rotated rx -180 ry 0 rz 65.72 deg; joints [-4.04, -53.566, 140.579, -182.534, 74.315, 90.059, 102.964]
  MoveL 1692 to (-203.17, 46.83, -10.48) mm, rotated rx 180 ry 0 rz 65.7 deg; joints [-4.04, -53.587, 140.582, -182.534, 74.298, 90.059, 102.979]
  MoveL 1693 to (222.09, 46.83, -10.48) mm, rotated rx 180 ry 0 rz -49.41 deg; joints [-4.281, -87.745, 145.701, -195.068, 6.349, 102.765, 179]
  MoveL 1694 to (223.29, 46.83, -10.47) mm, rotated rx -180 ry 0 rz -49.48 deg; joints [-4.284, -87.824, 145.757, -195.264, 6.266, 102.959, 179]
  MoveL 1695 to (223.53, 46.84, -10.47) mm, rotated rx 180 ry 0 rz -49.49 deg; joints [-4.285, -87.839, 145.77, -195.291, 6.255, 102.985, 179]
  MoveL 1696 to (223.77, 46.87, -10.48) mm, rotated rx -180 ry 0 rz -49.49 deg; joints [-4.285, -87.853, 145.786, -195.3, 6.252, 102.993, 179]
  MoveL 1697 to (224.01, 46.92, -10.48) mm, rotated rx -180 ry 0 rz -49.49 deg; joints [-4.286, -87.866, 145.803, -195.292, 6.258, 102.984, 179]
  MoveL 1698 to (224.24, 46.99, -10.48) mm, rotated rx 180 ry 0 rz -49.49 deg; joints [-4.287, -87.876, 145.822, -195.266, 6.27, 102.958, 179]
  MoveL 1699 to (224.46, 47.08, -10.48) mm, rotated rx 180 ry 0 rz -49.48 deg; joints [-4.287, -87.886, 145.844, -195.223, 6.291, 102.914, 179]
  MoveL 1700 to (224.69, 47.18, -10.48) mm, rotated rx -180 ry 0 rz -49.46 deg; joints [-4.288, -87.895, 145.868, -195.162, 6.32, 102.852, 179]
  MoveL 1701 to (224.92, 47.31, -10.48) mm, rotated rx 180 ry 0 rz -49.44 deg; joints [-4.289, -87.902, 145.895, -195.081, 6.359, 102.77, 179]
  MoveL 1702 to (225.07, 47.42, -10.48) mm, rotated rx -180 ry 0 rz -49.42 deg; joints [-4.29, -87.906, 145.916, -195.01, 6.393, 102.699, 179]
  MoveL 1703 to (225.23, 47.54, -10.48) mm, rotated rx 180 ry 0 rz -49.4 deg; joints [-4.291, -87.909, 145.939, -194.928, 6.432, 102.616, 179]
  MoveL 1704 to (225.39, 47.67, -10.47) mm, rotated rx 180 ry 0 rz -49.38 deg; joints [-4.292, -87.911, 145.964, -194.831, 6.479, 102.518, 179]
  MoveL 1705 to (225.55, 47.83, -10.48) mm, rotated rx -180 ry 0 rz -49.35 deg; joints [-4.293, -87.912, 145.991, -194.719, 6.535, 102.406, 179]
  MoveL 1706 to (225.66, 47.96, -10.47) mm, rotated rx 180 ry 0 rz -49.32 deg; joints [-4.293, -87.911, 146.013, -194.625, 6.581, 102.311, 179]
  MoveL 1707 to (225.77, 48.09, -10.48) mm, rotated rx 180 ry 0 rz -49.3 deg; joints [-4.294, -87.91, 146.035, -194.531, 6.629, 102.217, 179]
  MoveL 1708 to (225.86, 48.22, -10.48) mm, rotated rx -180 ry 0 rz -49.27 deg; joints [-4.295, -87.908, 146.056, -194.437, 6.677, 102.122, 179]
  MoveL 1709 to (225.94, 48.35, -10.47) mm, rotated rx -180 ry 0 rz -49.24 deg; joints [-4.295, -87.906, 146.076, -194.343, 6.726, 102.027, 179]
  MoveL 1710 to (226.07, 48.57, -10.48) mm, rotated rx -180 ry 0 rz -49.19 deg; joints [-4.296, -87.9, 146.11, -194.182, 6.812, 101.866, 179]
  MoveL 1711 to (226.17, 48.8, -10.48) mm, rotated rx -180 ry 0 rz -49.15 deg; joints [-4.297, -87.893, 146.143, -194.023, 6.898, 101.705, 179]
  MoveL 1712 to (226.25, 49.02, -10.48) mm, rotated rx -180 ry 0 rz -49.1 deg; joints [-4.298, -87.885, 146.175, -193.864, 6.987, 101.546, 179]
  MoveL 1713 to (226.31, 49.24, -10.48) mm, rotated rx 180 ry 0 rz -49.04 deg; joints [-4.299, -87.875, 146.207, -193.708, 7.076, 101.389, 179]
  MoveL 1714 to (226.36, 49.48, -10.47) mm, rotated rx -180 ry 0 rz -48.99 deg; joints [-4.3, -87.863, 146.24, -193.54, 7.175, 101.22, 179]
  MoveL 1715 to (226.39, 49.73, -10.48) mm, rotated rx -180 ry 0 rz -48.93 deg; joints [-4.301, -87.849, 146.272, -193.374, 7.275, 101.053, 179]
  MoveL 1716 to (226.4, 50.21, -10.48) mm, rotated rx 180 ry 0 rz -48.82 deg; joints [-4.303, -87.819, 146.333, -193.049, 7.478, 100.727, 179]
  MoveL 1717 to (226.4, 427.53, -10.47) mm, rotated rx -180 ry 0 rz -39.22 deg; joints [-4.514, -49.141, 151.053, -182.518, 60.294, 89.205, 179]
  MoveL 1718 to (226.39, 427.77, -10.48) mm, rotated rx -180 ry 0 rz -39.21 deg; joints [-4.514, -49.108, 151.049, -182.518, 60.337, 89.204, 179]
  MoveL 1719 to (226.37, 428.01, -10.48) mm, rotated rx -180 ry 0 rz -39.19 deg; joints [-4.515, -49.075, 151.044, -182.518, 60.383, 89.202, 179]
  MoveL 1720 to (226.34, 428.16, -10.48) mm, rotated rx -180 ry 0 rz -39.18 deg; joints [-4.515, -49.054, 151.041, -182.518, 60.411, 89.201, 179]
  MoveL 1721 to (226.31, 428.3, -10.48) mm, rotated rx 180 ry 0 rz -39.17 deg; joints [-4.515, -49.033, 151.037, -182.517, 60.44, 89.201, 179]
  MoveL 1722 to (226.27, 428.45, -10.48) mm, rotated rx 180 ry 0 rz -39.16 deg; joints [-4.515, -49.011, 151.033, -182.517, 60.469, 89.2, 179]
  MoveL 1723 to (226.22, 428.59, -10.48) mm, rotated rx 180 ry 0 rz -39.15 deg; joints [-4.515, -48.989, 151.029, -182.517, 60.5, 89.199, 179]
  MoveL 1724 to (226.16, 428.74, -10.48) mm, rotated rx -180 ry 0 rz -39.13 deg; joints [-4.515, -48.967, 151.024, -182.517, 60.531, 89.198, 179]
  MoveL 1725 to (226.1, 428.89, -10.48) mm, rotated rx -180 ry 0 rz -39.12 deg; joints [-4.515, -48.944, 151.019, -182.517, 60.563, 89.197, 179]
  MoveL 1726 to (226.03, 429.03, -10.48) mm, rotated rx 180 ry 0 rz -39.1 deg; joints [-4.515, -48.921, 151.013, -182.517, 60.596, 89.197, 179]
  MoveL 1727 to (225.94, 429.18, -10.48) mm, rotated rx -180 ry 0 rz -39.09 deg; joints [-4.515, -48.898, 151.006, -182.516, 60.63, 89.196, 179]
  MoveL 1728 to (225.82, 429.37, -10.48) mm, rotated rx -180 ry 0 rz -39.06 deg; joints [-4.515, -48.866, 150.997, -182.516, 60.677, 89.195, 179]
  MoveL 1729 to (225.67, 429.56, -10.48) mm, rotated rx 180 ry 0 rz -39.04 deg; joints [-4.515, -48.833, 150.987, -182.516, 60.725, 89.194, 179]
  MoveL 1730 to (225.5, 429.75, -10.48) mm, rotated rx -180 ry 0 rz -39.01 deg; joints [-4.515, -48.798, 150.975, -182.516, 60.776, 89.193, 179]
  MoveL 1731 to (225.29, 429.94, -10.48) mm, rotated rx 180 ry 0 rz -38.97 deg; joints [-4.514, -48.762, 150.962, -182.515, 60.831, 89.192, 179]
  MoveL 1732 to (225.13, 430.07, -10.47) mm, rotated rx 180 ry 0 rz -38.95 deg; joints [-4.514, -48.737, 150.951, -182.515, 60.869, 89.192, 179]
  MoveL 1733 to (224.97, 430.18, -10.48) mm, rotated rx -180 ry 0 rz -38.93 deg; joints [-4.514, -48.714, 150.941, -182.515, 60.905, 89.191, 179]
  MoveL 1734 to (224.81, 430.28, -10.48) mm, rotated rx -180 ry 0 rz -38.91 deg; joints [-4.514, -48.693, 150.931, -182.515, 60.938, 89.191, 179]
  MoveL 1735 to (224.65, 430.37, -10.48) mm, rotated rx 180 ry 0 rz -38.88 deg; joints [-4.513, -48.674, 150.922, -182.515, 60.97, 89.191, 179]
  MoveL 1736 to (224.49, 430.44, -10.48) mm, rotated rx -180 ry 0 rz -38.86 deg; joints [-4.513, -48.656, 150.912, -182.515, 60.999, 89.191, 179]
  MoveL 1737 to (224.33, 430.51, -10.47) mm, rotated rx -180 ry 0 rz -38.84 deg; joints [-4.513, -48.639, 150.903, -182.515, 61.026, 89.191, 179]
  MoveL 1738 to (224.17, 430.56, -10.48) mm, rotated rx -180 ry 0 rz -38.82 deg; joints [-4.513, -48.624, 150.894, -182.515, 61.052, 89.19, 179]
  MoveL 1739 to (224.01, 430.6, -10.48) mm, rotated rx -180 ry 0 rz -38.81 deg; joints [-4.512, -48.61, 150.885, -182.515, 61.076, 89.19, 179]
  MoveL 1740 to (223.77, 430.66, -10.48) mm, rotated rx -180 ry 0 rz -38.78 deg; joints [-4.512, -48.591, 150.871, -182.515, 61.11, 89.19, 179]
  MoveL 1741 to (223.53, 430.69, -10.48) mm, rotated rx -180 ry 0 rz -38.75 deg; joints [-4.512, -48.574, 150.858, -182.515, 61.14, 89.191, 179]
  MoveL 1742 to (223.29, 430.7, -10.48) mm, rotated rx -180 ry 0 rz -38.72 deg; joints [-4.511, -48.56, 150.845, -182.515, 61.167, 89.191, 179]
  MoveL 1743 to (223.05, 430.7, -10.48) mm, rotated rx 180 ry 0 rz -38.7 deg; joints [-4.511, -48.548, 150.832, -182.515, 61.192, 89.191, 179]
  MoveL 1744 to (-164.9, 430.7, -10.47) mm, rotated rx 180 ry 0 rz 9.63 deg; joints [-4.073, -32.14, 134.47, -182.472, 89.618, 89.382, 159.05]
  Set speed (38.1 mm/s)
  MoveL 1745 to (-165.25, 431.87, -10.48) mm, rotated rx 180 ry 0 rz 9.62 deg; joints [-4.073, -32.041, 134.427, -182.472, 89.674, 89.38, 159.061]
  MoveL 1746 to (-164.27, 432.52, -10.48) mm, rotated rx 180 ry 0 rz 9.48 deg; joints [-4.073, -32.02, 134.418, -182.472, 89.686, 89.379, 159.204]
  Set speed (25.4 mm/s)
  MoveL 1747 to (-164.27, 432.52, -12.84) mm, rotated rx -180 ry 0 rz 9.48 deg; joints [-4.203, -32.021, 134.41, -182.599, 89.677, 89.352, 159.204]
  MoveL 1748 to (-164.27, 431.89, -13.47) mm, rotated rx 180 ry 0 rz 9.5 deg; joints [-4.238, -32.069, 134.43, -182.633, 89.647, 89.346, 159.176]
  Set speed (38.1 mm/s)
  MoveL 1749 to (-164.9, 431.25, -13.47) mm, rotated rx -180 ry 0 rz 9.61 deg; joints [-4.238, -32.099, 134.443, -182.633, 89.63, 89.346, 159.074]
  Set speed (76.2 mm/s)
  MoveL 1750 to (-194.97, 431.25, -13.47) mm, rotated rx 180 ry 0 rz 13.01 deg; joints [-4.24, -31.156, 134.024, -182.635, 90.154, 89.322, 155.672]
  MoveL 1751 to (-201.24, 431.25, -13.48) mm, rotated rx 180 ry 0 rz 13.7 deg; joints [-4.24, -30.944, 133.928, -182.635, 90.27, 89.317, 154.985]
  MoveL 1752 to (-201.48, 431.25, -13.48) mm, rotated rx 180 ry 0 rz 13.72 deg; joints [-4.24, -30.936, 133.924, -182.635, 90.275, 89.316, 154.958]
  MoveL 1753 to (-201.72, 431.23, -13.48) mm, rotated rx 180 ry 0 rz 13.75 deg; joints [-4.24, -30.929, 133.921, -182.635, 90.278, 89.316, 154.931]
  MoveL 1754 to (-201.96, 431.19, -13.48) mm, rotated rx 180 ry 0 rz 13.78 deg; joints [-4.24, -30.923, 133.919, -182.635, 90.281, 89.316, 154.902]
  MoveL 1755 to (-202.2, 431.13, -13.48) mm, rotated rx 180 ry 0 rz 13.81 deg; joints [-4.24, -30.919, 133.917, -182.635, 90.283, 89.316, 154.873]
  MoveL 1756 to (-204.13, 430.52, -13.47) mm, rotated rx 180 ry 0 rz 14.05 deg; joints [-4.24, -30.897, 133.907, -182.635, 90.295, 89.315, 154.632]
  MoveL 1757 to (-204.42, 430.43, -13.48) mm, rotated rx -180 ry 0 rz 14.08 deg; joints [-4.24, -30.894, 133.905, -182.635, 90.297, 89.315, 154.595]
  MoveL 1758 to (-204.57, 430.37, -13.48) mm, rotated rx -180 ry 0 rz 14.1 deg; joints [-4.24, -30.893, 133.905, -182.635, 90.298, 89.315, 154.577]
  MoveL 1759 to (-204.72, 430.31, -13.48) mm, rotated rx 180 ry 0 rz 14.12 deg; joints [-4.24, -30.893, 133.905, -182.635, 90.298, 89.315, 154.557]
  MoveL 1760 to (-204.86, 430.23, -13.48) mm, rotated rx 180 ry 0 rz 14.14 deg; joints [-4.24, -30.893, 133.905, -182.635, 90.298, 89.315, 154.538]
  MoveL 1761 to (-205.01, 430.15, -13.47) mm, rotated rx -180 ry 0 rz 14.16 deg; joints [-4.24, -30.894, 133.906, -182.635, 90.297, 89.315, 154.517]
  MoveL 1762 to (-205.16, 430.05, -13.47) mm, rotated rx 180 ry 0 rz 14.18 deg; joints [-4.24, -30.896, 133.906, -182.635, 90.296, 89.315, 154.497]
  MoveL 1763 to (-205.3, 429.94, -13.48) mm, rotated rx -180 ry 0 rz 14.2 deg; joints [-4.24, -30.899, 133.908, -182.635, 90.294, 89.315, 154.475]
  MoveL 1764 to (-205.53, 429.75, -13.47) mm, rotated rx 180 ry 0 rz 14.24 deg; joints [-4.24, -30.905, 133.911, -182.635, 90.291, 89.316, 154.441]
  MoveL 1765 to (-205.75, 429.52, -13.47) mm, rotated rx 180 ry 0 rz 14.28 deg; joints [-4.24, -30.914, 133.915, -182.635, 90.286, 89.316, 154.404]
  MoveL 1766 to (-205.92, 429.3, -13.48) mm, rotated rx 180 ry 0 rz 14.3 deg; joints [-4.24, -30.924, 133.919, -182.635, 90.281, 89.316, 154.375]
  MoveL 1767 to (-206.06, 429.09, -13.48) mm, rotated rx 180 ry 0 rz 14.33 deg; joints [-4.24, -30.935, 133.924, -182.635, 90.275, 89.316, 154.348]
  MoveL 1768 to (-206.14, 428.95, -13.48) mm, rotated rx 180 ry 0 rz 14.35 deg; joints [-4.24, -30.942, 133.927, -182.635, 90.271, 89.316, 154.333]
  MoveL 1769 to (-206.21, 428.82, -13.48) mm, rotated rx 180 ry 0 rz 14.36 deg; joints [-4.24, -30.949, 133.931, -182.635, 90.267, 89.317, 154.319]
  MoveL 1770 to (-206.27, 428.69, -13.48) mm, rotated rx 180 ry 0 rz 14.37 deg; joints [-4.24, -30.957, 133.934, -182.635, 90.263, 89.317, 154.305]
  MoveL 1771 to (-206.32, 428.55, -13.48) mm, rotated rx 180 ry 0 rz 14.39 deg; joints [-4.24, -30.965, 133.938, -182.635, 90.258, 89.317, 154.292]
  MoveL 1772 to (-206.37, 428.42, -13.47) mm, rotated rx 180 ry 0 rz 14.4 deg; joints [-4.24, -30.973, 133.941, -182.635, 90.254, 89.317, 154.28]
  MoveL 1773 to (-206.41, 428.28, -13.47) mm, rotated rx 180 ry 0 rz 14.41 deg; joints [-4.24, -30.982, 133.945, -182.635, 90.249, 89.318, 154.268]
  MoveL 1774 to (-206.47, 428.01, -13.48) mm, rotated rx 180 ry 0 rz 14.43 deg; joints [-4.24, -30.999, 133.953, -182.635, 90.24, 89.318, 154.248]
  MoveL 1775 to (-206.5, 427.77, -13.48) mm, rotated rx 180 ry 0 rz 14.45 deg; joints [-4.24, -31.016, 133.961, -182.635, 90.231, 89.318, 154.231]
  MoveL 1776 to (-206.52, 427.53, -13.47) mm, rotated rx 180 ry 0 rz 14.46 deg; joints [-4.24, -31.033, 133.968, -182.635, 90.221, 89.319, 154.217]
  MoveL 1777 to (-206.52, 427.04, -13.48) mm, rotated rx -180 ry 0 rz 14.49 deg; joints [-4.24, -31.068, 133.984, -182.635, 90.202, 89.32, 154.191]
  MoveL 1778 to (-206.52, 50.21, -13.47) mm, rotated rx 180 ry 0 rz 65.02 deg; joints [-4.205, -53.237, 140.523, -182.698, 74.589, 90.054, 103.664]
  MoveL 1779 to (-206.51, 49.73, -13.47) mm, rotated rx 180 ry 0 rz 65.14 deg; joints [-4.205, -53.248, 140.525, -182.698, 74.58, 90.055, 103.539]
  MoveL 1780 to (-206.48, 49.48, -13.48) mm, rotated rx -180 ry 0 rz 65.2 deg; joints [-4.205, -53.255, 140.526, -182.698, 74.574, 90.055, 103.477]
  MoveL 1781 to (-206.43, 49.24, -13.47) mm, rotated rx 180 ry 0 rz 65.26 deg; joints [-4.205, -53.264, 140.527, -182.698, 74.566, 90.055, 103.417]
  MoveL 1782 to (-206.37, 49.02, -13.47) mm, rotated rx -180 ry 0 rz 65.32 deg; joints [-4.205, -53.274, 140.528, -182.698, 74.557, 90.056, 103.362]
  MoveL 1783 to (-206.28, 48.8, -13.47) mm, rotated rx 180 ry 0 rz 65.37 deg; joints [-4.205, -53.285, 140.53, -182.698, 74.548, 90.056, 103.309]
  MoveL 1784 to (-206.18, 48.57, -13.47) mm, rotated rx 180 ry 0 rz 65.42 deg; joints [-4.205, -53.298, 140.532, -182.698, 74.537, 90.057, 103.256]
  MoveL 1785 to (-206.06, 48.35, -13.48) mm, rotated rx -180 ry 0 rz 65.47 deg; joints [-4.205, -53.312, 140.534, -182.699, 74.524, 90.057, 103.205]
  MoveL 1786 to (-205.98, 48.22, -13.47) mm, rotated rx 180 ry 0 rz 65.5 deg; joints [-4.205, -53.322, 140.535, -182.699, 74.516, 90.058, 103.176]
  MoveL 1787 to (-205.88, 48.09, -13.48) mm, rotated rx -180 ry 0 rz 65.53 deg; joints [-4.205, -53.332, 140.537, -182.699, 74.507, 90.058, 103.148]
  MoveL 1788 to (-205.78, 47.96, -13.47) mm, rotated rx 180 ry 0 rz 65.56 deg; joints [-4.205, -53.344, 140.538, -182.699, 74.497, 90.059, 103.12]
  MoveL 1789 to (-205.66, 47.83, -13.48) mm, rotated rx -180 ry 0 rz 65.59 deg; joints [-4.205, -53.356, 140.54, -182.699, 74.487, 90.059, 103.092]
  MoveL 1790 to (-205.51, 47.67, -13.47) mm, rotated rx 180 ry 0 rz 65.62 deg; joints [-4.205, -53.372, 140.542, -182.699, 74.473, 90.06, 103.06]
  MoveL 1791 to (-205.35, 47.54, -13.48) mm, rotated rx -180 ry 0 rz 65.65 deg; joints [-4.205, -53.388, 140.544, -182.699, 74.459, 90.061, 103.034]
  MoveL 1792 to (-205.19, 47.42, -13.47) mm, rotated rx 180 ry 0 rz 65.67 deg; joints [-4.205, -53.403, 140.547, -182.699, 74.446, 90.061, 103.012]
  MoveL 1793 to (-205.03, 47.31, -13.48) mm, rotated rx 180 ry 0 rz 65.69 deg; joints [-4.205, -53.419, 140.549, -182.7, 74.433, 90.062, 102.993]
  MoveL 1794 to (-204.81, 47.18, -13.48) mm, rotated rx -180 ry 0 rz 65.71 deg; joints [-4.205, -53.44, 140.552, -182.7, 74.415, 90.063, 102.973]
  MoveL 1795 to (-204.58, 47.08, -13.47) mm, rotated rx 180 ry 0 rz 65.72 deg; joints [-4.205, -53.461, 140.555, -182.7, 74.397, 90.064, 102.958]
  MoveL 1796 to (-204.36, 46.99, -13.47) mm, rotated rx 180 ry 0 rz 65.73 deg; joints [-4.205, -53.482, 140.558, -182.7, 74.379, 90.064, 102.95]
  MoveL 1797 to (-204.13, 46.92, -13.47) mm, rotated rx 180 ry 0 rz 65.73 deg; joints [-4.205, -53.502, 140.56, -182.7, 74.362, 90.065, 102.946]
  MoveL 1798 to (-203.89, 46.87, -13.47) mm, rotated rx 180 ry 0 rz 65.73 deg; joints [-4.204, -53.523, 140.563, -182.701, 74.343, 90.066, 102.947]
  MoveL 1799 to (-203.65, 46.84, -13.48) mm, rotated rx 180 ry 0 rz 65.73 deg; joints [-4.204, -53.544, 140.566, -182.701, 74.325, 90.067, 102.953]
  MoveL 1800 to (-203.41, 46.83, -13.48) mm, rotated rx 180 ry 0 rz 65.72 deg; joints [-4.204, -53.564, 140.569, -182.701, 74.308, 90.068, 102.964]
  MoveL 1801 to (-203.17, 46.83, -13.48) mm, rotated rx 180 ry 0 rz 65.7 deg; joints [-4.204, -53.584, 140.572, -182.701, 74.29, 90.069, 102.979]
  MoveL 1802 to (222.09, 46.83, -13.48) mm, rotated rx 180 ry 0 rz -49.41 deg; joints [-4.464, -87.736, 145.691, -196.061, 6.374, 103.608, 179]
  MoveL 1803 to (223.29, 46.83, -13.47) mm, rotated rx -180 ry 0 rz -49.48 deg; joints [-4.466, -87.815, 145.747, -196.269, 6.291, 103.814, 179]
  MoveL 1804 to (223.53, 46.84, -13.48) mm, rotated rx 180 ry 0 rz -49.49 deg; joints [-4.467, -87.83, 145.76, -196.297, 6.281, 103.841, 179]
  MoveL 1805 to (223.77, 46.87, -13.47) mm, rotated rx 180 ry 0 rz -49.49 deg; joints [-4.468, -87.843, 145.775, -196.307, 6.278, 103.85, 179]
  MoveL 1806 to (224.01, 46.92, -13.48) mm, rotated rx 180 ry 0 rz -49.49 deg; joints [-4.469, -87.856, 145.793, -196.298, 6.283, 103.84, 179]
  MoveL 1807 to (224.24, 46.99, -13.48) mm, rotated rx -180 ry 0 rz -49.49 deg; joints [-4.469, -87.867, 145.812, -196.271, 6.296, 103.813, 179]
  MoveL 1808 to (224.46, 47.08, -13.47) mm, rotated rx 180 ry 0 rz -49.48 deg; joints [-4.47, -87.877, 145.834, -196.226, 6.316, 103.767, 179]
  MoveL 1809 to (224.69, 47.18, -13.47) mm, rotated rx -180 ry 0 rz -49.46 deg; joints [-4.471, -87.885, 145.858, -196.16, 6.345, 103.701, 179]
  MoveL 1810 to (224.92, 47.31, -13.48) mm, rotated rx 180 ry 0 rz -49.44 deg; joints [-4.472, -87.892, 145.885, -196.074, 6.384, 103.613, 179]
  MoveL 1811 to (225.07, 47.42, -13.47) mm, rotated rx -180 ry 0 rz -49.42 deg; joints [-4.473, -87.896, 145.906, -195.999, 6.418, 103.538, 179]
  MoveL 1812 to (225.23, 47.54, -13.47) mm, rotated rx 180 ry 0 rz -49.4 deg; joints [-4.474, -87.899, 145.928, -195.912, 6.457, 103.45, 179]
  MoveL 1813 to (225.39, 47.67, -13.48) mm, rotated rx 180 ry 0 rz -49.38 deg; joints [-4.475, -87.901, 145.953, -195.809, 6.504, 103.347, 179]
  MoveL 1814 to (225.55, 47.83, -13.48) mm, rotated rx -180 ry 0 rz -49.35 deg; joints [-4.476, -87.902, 145.981, -195.691, 6.559, 103.227, 179]
  MoveL 1815 to (225.66, 47.96, -13.48) mm, rotated rx -180 ry 0 rz -49.32 deg; joints [-4.476, -87.902, 146.003, -195.591, 6.606, 103.127, 179]
  MoveL 1816 to (225.77, 48.09, -13.47) mm, rotated rx -180 ry 0 rz -49.3 deg; joints [-4.477, -87.901, 146.024, -195.491, 6.653, 103.027, 179]
  MoveL 1817 to (225.86, 48.22, -13.48) mm, rotated rx -180 ry 0 rz -49.27 deg; joints [-4.478, -87.899, 146.045, -195.391, 6.701, 102.926, 179]
  MoveL 1818 to (225.94, 48.35, -13.47) mm, rotated rx -180 ry 0 rz -49.24 deg; joints [-4.479, -87.896, 146.066, -195.292, 6.75, 102.826, 179]
  MoveL 1819 to (226.07, 48.57, -13.47) mm, rotated rx -180 ry 0 rz -49.19 deg; joints [-4.48, -87.891, 146.1, -195.121, 6.835, 102.654, 179]
  MoveL 1820 to (226.17, 48.8, -13.48) mm, rotated rx 180 ry 0 rz -49.15 deg; joints [-4.481, -87.884, 146.133, -194.952, 6.922, 102.484, 179]
  MoveL 1821 to (226.25, 49.02, -13.47) mm, rotated rx 180 ry 0 rz -49.1 deg; joints [-4.482, -87.875, 146.165, -194.784, 7.01, 102.315, 179]
  MoveL 1822 to (226.31, 49.24, -13.47) mm, rotated rx 180 ry 0 rz -49.04 deg; joints [-4.483, -87.865, 146.196, -194.617, 7.099, 102.148, 179]
  MoveL 1823 to (226.36, 49.48, -13.47) mm, rotated rx -180 ry 0 rz -48.99 deg; joints [-4.484, -87.853, 146.229, -194.438, 7.197, 101.968, 179]
  MoveL 1824 to (226.39, 49.73, -13.48) mm, rotated rx -180 ry 0 rz -48.93 deg; joints [-4.485, -87.84, 146.261, -194.262, 7.297, 101.791, 179]
  MoveL 1825 to (226.4, 50.21, -13.48) mm, rotated rx -180 ry 0 rz -48.82 deg; joints [-4.487, -87.81, 146.323, -193.917, 7.499, 101.445, 179]
  MoveL 1826 to (226.4, 428.01, -13.47) mm, rotated rx -180 ry 0 rz -39.2 deg; joints [-4.71, -49.078, 151.035, -182.686, 60.365, 89.156, 179]
  MoveL 1827 to (226.4, 428.22, -13.47) mm, rotated rx -180 ry 0 rz -39.19 deg; joints [-4.71, -49.049, 151.032, -182.686, 60.403, 89.155, 179]
  MoveL 1828 to (226.38, 428.44, -13.48) mm, rotated rx -180 ry 0 rz -39.17 deg; joints [-4.71, -49.019, 151.029, -182.686, 60.442, 89.154, 179]
  MoveL 1829 to (226.35, 428.65, -13.48) mm, rotated rx -180 ry 0 rz -39.16 deg; joints [-4.711, -48.989, 151.024, -182.685, 60.483, 89.152, 179]
  MoveL 1830 to (226.3, 428.87, -13.48) mm, rotated rx -180 ry 0 rz -39.14 deg; joints [-4.711, -48.958, 151.019, -182.685, 60.526, 89.151, 179]
  MoveL 1831 to (226.24, 429.08, -13.47) mm, rotated rx 180 ry 0 rz -39.12 deg; joints [-4.711, -48.926, 151.013, -182.685, 60.57, 89.15, 179]
  MoveL 1832 to (226.16, 429.3, -13.48) mm, rotated rx -180 ry 0 rz -39.1 deg; joints [-4.711, -48.894, 151.006, -182.684, 60.615, 89.149, 179]
  MoveL 1833 to (226.06, 429.51, -13.47) mm, rotated rx 180 ry 0 rz -39.08 deg; joints [-4.711, -48.86, 150.997, -182.684, 60.663, 89.147, 179]
  MoveL 1834 to (225.94, 429.73, -13.48) mm, rotated rx -180 ry 0 rz -39.05 deg; joints [-4.711, -48.825, 150.988, -182.684, 60.713, 89.146, 179]
  MoveL 1835 to (225.8, 429.94, -13.47) mm, rotated rx -180 ry 0 rz -39.03 deg; joints [-4.711, -48.789, 150.978, -182.684, 60.765, 89.145, 179]
  MoveL 1836 to (225.6, 430.19, -13.48) mm, rotated rx -180 ry 0 rz -38.99 deg; joints [-4.711, -48.746, 150.964, -182.683, 60.829, 89.144, 179]
  MoveL 1837 to (225.35, 430.44, -13.48) mm, rotated rx -180 ry 0 rz -38.95 deg; joints [-4.71, -48.701, 150.947, -182.683, 60.897, 89.143, 179]
  MoveL 1838 to (225.13, 430.62, -13.48) mm, rotated rx -180 ry 0 rz -38.92 deg; joints [-4.71, -48.665, 150.933, -182.683, 60.951, 89.142, 179]
  MoveL 1839 to (224.91, 430.77, -13.48) mm, rotated rx -180 ry 0 rz -38.89 deg; joints [-4.71, -48.633, 150.919, -182.683, 61.001, 89.141, 179]
  MoveL 1840 to (224.68, 430.9, -13.47) mm, rotated rx -180 ry 0 rz -38.86 deg; joints [-4.709, -48.605, 150.905, -182.682, 61.045, 89.141, 179]
  MoveL 1841 to (224.46, 431, -13.48) mm, rotated rx 180 ry 0 rz -38.83 deg; joints [-4.709, -48.58, 150.892, -182.682, 61.086, 89.141, 179]
  MoveL 1842 to (224.24, 431.09, -13.48) mm, rotated rx -180 ry 0 rz -38.8 deg; joints [-4.709, -48.558, 150.879, -182.682, 61.123, 89.14, 179]
  MoveL 1843 to (224.01, 431.15, -13.48) mm, rotated rx 180 ry 0 rz -38.78 deg; joints [-4.708, -48.538, 150.866, -182.682, 61.157, 89.14, 179]
  MoveL 1844 to (223.77, 431.21, -13.48) mm, rotated rx -180 ry 0 rz -38.75 deg; joints [-4.708, -48.519, 150.852, -182.682, 61.191, 89.14, 179]
  MoveL 1845 to (223.53, 431.24, -13.48) mm, rotated rx -180 ry 0 rz -38.72 deg; joints [-4.707, -48.502, 150.839, -182.682, 61.221, 89.141, 179]
  MoveL 1846 to (223.29, 431.25, -13.48) mm, rotated rx 180 ry 0 rz -38.69 deg; joints [-4.707, -48.488, 150.826, -182.682, 61.248, 89.141, 179]
  MoveL 1847 to (223.05, 431.25, -13.48) mm, rotated rx -180 ry 0 rz -38.67 deg; joints [-4.706, -48.476, 150.813, -182.682, 61.273, 89.141, 179]
  MoveL 1848 to (-164.9, 431.25, -13.48) mm, rotated rx 180 ry 0 rz 9.61 deg; joints [-4.238, -32.099, 134.443, -182.633, 89.63, 89.346, 159.074]
  Set speed (38.1 mm/s)
  MoveL 1849 to (-165.25, 432.42, -13.48) mm, rotated rx -180 ry 0 rz 9.59 deg; joints [-4.239, -32, 134.399, -182.634, 89.686, 89.344, 159.085]
  MoveL 1850 to (-164.27, 433.07, -13.48) mm, rotated rx -180 ry 0 rz 9.45 deg; joints [-4.239, -31.979, 134.39, -182.634, 89.698, 89.343, 159.228]
  Set speed (25.4 mm/s)
  MoveL 1851 to (-164.27, 433.07, -15.84) mm, rotated rx -180 ry 0 rz 9.45 deg; joints [-4.369, -31.979, 134.382, -182.761, 89.688, 89.316, 159.228]
  MoveL 1852 to (-164.27, 432.44, -16.48) mm, rotated rx 180 ry 0 rz 9.48 deg; joints [-4.404, -32.028, 134.402, -182.795, 89.658, 89.31, 159.2]
  Set speed (38.1 mm/s)
  MoveL 1853 to (-164.9, 431.8, -16.48) mm, rotated rx 180 ry 0 rz 9.58 deg; joints [-4.404, -32.058, 134.415, -182.795, 89.641, 89.31, 159.098]
  Set speed (76.2 mm/s)
  MoveL 1854 to (-194.97, 431.8, -16.48) mm, rotated rx -180 ry 0 rz 12.98 deg; joints [-4.406, -31.116, 133.996, -182.797, 90.164, 89.285, 155.7]
  MoveL 1855 to (-199.31, 431.8, -16.48) mm, rotated rx 180 ry 0 rz 13.46 deg; joints [-4.406, -30.97, 133.93, -182.797, 90.244, 89.281, 155.223]
  MoveL 1856 to (-199.79, 431.8, -16.48) mm, rotated rx -180 ry 0 rz 13.51 deg; joints [-4.406, -30.954, 133.923, -182.797, 90.253, 89.28, 155.17]
  MoveL 1857 to (-200.03, 431.77, -16.47) mm, rotated rx 180 ry 0 rz 13.54 deg; joints [-4.406, -30.948, 133.92, -182.797, 90.256, 89.28, 155.142]
  MoveL 1858 to (-200.27, 431.73, -16.48) mm, rotated rx -180 ry 0 rz 13.57 deg; joints [-4.406, -30.943, 133.917, -182.797, 90.259, 89.28, 155.114]
  MoveL 1859 to (-200.52, 431.67, -16.47) mm, rotated rx -180 ry 0 rz 13.6 deg; joints [-4.406, -30.939, 133.916, -182.797, 90.261, 89.28, 155.084]
  MoveL 1860 to (-204.13, 430.52, -16.48) mm, rotated rx 180 ry 0 rz 14.05 deg; joints [-4.406, -30.898, 133.897, -182.797, 90.283, 89.279, 154.632]
  MoveL 1861 to (-204.42, 430.43, -16.48) mm, rotated rx 180 ry 0 rz 14.08 deg; joints [-4.406, -30.895, 133.896, -182.797, 90.285, 89.279, 154.595]
  MoveL 1862 to (-204.57, 430.37, -16.48) mm, rotated rx -180 ry 0 rz 14.1 deg; joints [-4.406, -30.894, 133.895, -182.797, 90.285, 89.279, 154.577]
  MoveL 1863 to (-204.72, 430.31, -16.48) mm, rotated rx 180 ry 0 rz 14.12 deg; joints [-4.406, -30.894, 133.895, -182.797, 90.285, 89.278, 154.557]
  MoveL 1864 to (-204.86, 430.23, -16.47) mm, rotated rx -180 ry 0 rz 14.14 deg; joints [-4.406, -30.894, 133.895, -182.797, 90.285, 89.279, 154.538]
  MoveL 1865 to (-205.01, 430.15, -16.48) mm, rotated rx 180 ry 0 rz 14.16 deg; joints [-4.406, -30.895, 133.896, -182.797, 90.285, 89.279, 154.517]
  MoveL 1866 to (-205.16, 430.05, -16.47) mm, rotated rx 180 ry 0 rz 14.18 deg; joints [-4.406, -30.897, 133.897, -182.797, 90.284, 89.279, 154.497]
  MoveL 1867 to (-205.3, 429.94, -16.48) mm, rotated rx -180 ry 0 rz 14.2 deg; joints [-4.406, -30.9, 133.898, -182.797, 90.282, 89.279, 154.475]
  MoveL 1868 to (-205.53, 429.75, -16.47) mm, rotated rx -180 ry 0 rz 14.24 deg; joints [-4.406, -30.906, 133.901, -182.797, 90.279, 89.279, 154.441]
  MoveL 1869 to (-205.75, 429.52, -16.48) mm, rotated rx 180 ry 0 rz 14.28 deg; joints [-4.406, -30.915, 133.905, -182.797, 90.274, 89.279, 154.404]
  MoveL 1870 to (-205.92, 429.3, -16.48) mm, rotated rx -180 ry 0 rz 14.3 deg; joints [-4.406, -30.925, 133.91, -182.797, 90.268, 89.279, 154.375]
  MoveL 1871 to (-206.06, 429.09, -16.48) mm, rotated rx 180 ry 0 rz 14.33 deg; joints [-4.406, -30.936, 133.914, -182.797, 90.263, 89.28, 154.348]
  MoveL 1872 to (-206.14, 428.95, -16.47) mm, rotated rx 180 ry 0 rz 14.35 deg; joints [-4.406, -30.943, 133.918, -182.797, 90.259, 89.28, 154.333]
  MoveL 1873 to (-206.21, 428.82, -16.48) mm, rotated rx 180 ry 0 rz 14.36 deg; joints [-4.406, -30.95, 133.921, -182.797, 90.255, 89.28, 154.319]
  MoveL 1874 to (-206.27, 428.69, -16.47) mm, rotated rx 180 ry 0 rz 14.37 deg; joints [-4.406, -30.958, 133.924, -182.797, 90.25, 89.28, 154.305]
  MoveL 1875 to (-206.32, 428.55, -16.47) mm, rotated rx -180 ry 0 rz 14.39 deg; joints [-4.406, -30.966, 133.928, -182.797, 90.246, 89.28, 154.292]
  MoveL 1876 to (-206.37, 428.42, -16.47) mm, rotated rx 180 ry 0 rz 14.4 deg; joints [-4.406, -30.974, 133.932, -182.797, 90.242, 89.281, 154.28]
  MoveL 1877 to (-206.41, 428.28, -16.47) mm, rotated rx -180 ry 0 rz 14.41 deg; joints [-4.406, -30.983, 133.936, -182.797, 90.237, 89.281, 154.268]
  MoveL 1878 to (-206.47, 428.01, -16.47) mm, rotated rx -180 ry 0 rz 14.43 deg; joints [-4.406, -31, 133.944, -182.797, 90.227, 89.281, 154.248]
  MoveL 1879 to (-206.5, 427.77, -16.48) mm, rotated rx 180 ry 0 rz 14.45 deg; joints [-4.406, -31.017, 133.951, -182.797, 90.218, 89.282, 154.231]
  MoveL 1880 to (-206.52, 427.53, -16.47) mm, rotated rx -180 ry 0 rz 14.46 deg; joints [-4.406, -31.034, 133.959, -182.797, 90.209, 89.282, 154.217]
  MoveL 1881 to (-206.52, 427.04, -16.48) mm, rotated rx -180 ry 0 rz 14.49 deg; joints [-4.406, -31.069, 133.975, -182.797, 90.19, 89.283, 154.191]
  MoveL 1882 to (-206.52, 50.21, -16.48) mm, rotated rx -180 ry 0 rz 65.02 deg; joints [-4.37, -53.234, 140.513, -182.865, 74.581, 90.063, 103.664]
  MoveL 1883 to (-206.51, 49.73, -16.47) mm, rotated rx 180 ry 0 rz 65.14 deg; joints [-4.37, -53.245, 140.514, -182.865, 74.572, 90.063, 103.539]
  MoveL 1884 to (-206.48, 49.48, -16.47) mm, rotated rx 180 ry 0 rz 65.2 deg; joints [-4.37, -53.252, 140.515, -182.865, 74.566, 90.063, 103.477]
  MoveL 1885 to (-206.43, 49.24, -16.48) mm, rotated rx -180 ry 0 rz 65.26 deg; joints [-4.37, -53.261, 140.516, -182.865, 74.558, 90.064, 103.417]
  MoveL 1886 to (-206.37, 49.02, -16.48) mm, rotated rx -180 ry 0 rz 65.32 deg; joints [-4.37, -53.271, 140.518, -182.865, 74.55, 90.064, 103.362]
  MoveL 1887 to (-206.28, 48.8, -16.47) mm, rotated rx 180 ry 0 rz 65.37 deg; joints [-4.37, -53.282, 140.519, -182.865, 74.54, 90.065, 103.309]
  MoveL 1888 to (-206.18, 48.57, -16.48) mm, rotated rx -180 ry 0 rz 65.42 deg; joints [-4.37, -53.295, 140.521, -182.865, 74.529, 90.065, 103.256]
  MoveL 1889 to (-206.06, 48.35, -16.48) mm, rotated rx -180 ry 0 rz 65.47 deg; joints [-4.37, -53.31, 140.523, -182.865, 74.516, 90.066, 103.205]
  MoveL 1890 to (-205.98, 48.22, -16.48) mm, rotated rx 180 ry 0 rz 65.5 deg; joints [-4.37, -53.319, 140.525, -182.865, 74.508, 90.066, 103.176]
  MoveL 1891 to (-205.88, 48.09, -16.48) mm, rotated rx -180 ry 0 rz 65.53 deg; joints [-4.369, -53.33, 140.526, -182.866, 74.499, 90.067, 103.148]
  MoveL 1892 to (-205.78, 47.96, -16.47) mm, rotated rx -180 ry 0 rz 65.56 deg; joints [-4.369, -53.341, 140.528, -182.866, 74.49, 90.067, 103.12]
  MoveL 1893 to (-205.66, 47.83, -16.48) mm, rotated rx 180 ry 0 rz 65.59 deg; joints [-4.369, -53.353, 140.529, -182.866, 74.479, 90.068, 103.092]
  MoveL 1894 to (-205.51, 47.67, -16.48) mm, rotated rx -180 ry 0 rz 65.62 deg; joints [-4.369, -53.369, 140.532, -182.866, 74.465, 90.069, 103.06]
  MoveL 1895 to (-205.35, 47.54, -16.47) mm, rotated rx -180 ry 0 rz 65.65 deg; joints [-4.369, -53.385, 140.534, -182.866, 74.452, 90.069, 103.034]
  MoveL 1896 to (-205.19, 47.42, -16.47) mm, rotated rx 180 ry 0 rz 65.67 deg; joints [-4.369, -53.401, 140.536, -182.866, 74.438, 90.07, 103.012]
  MoveL 1897 to (-205.03, 47.31, -16.48) mm, rotated rx 180 ry 0 rz 65.69 deg; joints [-4.369, -53.416, 140.538, -182.866, 74.425, 90.071, 102.993]
  MoveL 1898 to (-204.81, 47.18, -16.48) mm, rotated rx 180 ry 0 rz 65.71 deg; joints [-4.369, -53.438, 140.541, -182.867, 74.407, 90.072, 102.973]
  MoveL 1899 to (-204.58, 47.08, -16.48) mm, rotated rx -180 ry 0 rz 65.72 deg; joints [-4.369, -53.458, 140.544, -182.867, 74.389, 90.073, 102.958]
  MoveL 1900 to (-204.36, 46.99, -16.47) mm, rotated rx 180 ry 0 rz 65.73 deg; joints [-4.369, -53.479, 140.547, -182.867, 74.371, 90.074, 102.95]
  MoveL 1901 to (-204.13, 46.92, -16.48) mm, rotated rx -180 ry 0 rz 65.73 deg; joints [-4.369, -53.499, 140.55, -182.867, 74.354, 90.074, 102.946]
  MoveL 1902 to (-203.89, 46.87, -16.48) mm, rotated rx 180 ry 0 rz 65.73 deg; joints [-4.369, -53.52, 140.553, -182.868, 74.336, 90.075, 102.947]
  MoveL 1903 to (-203.65, 46.84, -16.48) mm, rotated rx -180 ry 0 rz 65.73 deg; joints [-4.369, -53.541, 140.555, -182.868, 74.318, 90.076, 102.953]
  MoveL 1904 to (-203.41, 46.83, -16.48) mm, rotated rx -180 ry 0 rz 65.72 deg; joints [-4.369, -53.562, 140.558, -182.868, 74.3, 90.077, 102.964]
  MoveL 1905 to (-203.17, 46.83, -16.48) mm, rotated rx 180 ry 0 rz 65.7 deg; joints [-4.369, -53.582, 140.561, -182.868, 74.283, 90.078, 102.979]
  MoveL 1906 to (222.09, 46.83, -16.48) mm, rotated rx 180 ry 0 rz -49.41 deg; joints [-4.646, -87.726, 145.68, -197.046, 6.4, 104.444, 179]
  MoveL 1907 to (223.29, 46.83, -16.48) mm, rotated rx 180 ry 0 rz -49.48 deg; joints [-4.649, -87.805, 145.736, -197.266, 6.318, 104.661, 179]
  MoveL 1908 to (223.53, 46.84, -16.48) mm, rotated rx 180 ry 0 rz -49.49 deg; joints [-4.65, -87.82, 145.749, -197.296, 6.308, 104.69, 179]
  MoveL 1909 to (223.77, 46.87, -16.48) mm, rotated rx -180 ry 0 rz -49.49 deg; joints [-4.65, -87.833, 145.764, -197.306, 6.305, 104.7, 179]
  MoveL 1910 to (224.01, 46.92, -16.48) mm, rotated rx -180 ry 0 rz -49.49 deg; joints [-4.651, -87.846, 145.782, -197.296, 6.31, 104.689, 179]
  MoveL 1911 to (224.24, 46.99, -16.47) mm, rotated rx -180 ry 0 rz -49.49 deg; joints [-4.652, -87.857, 145.801, -197.268, 6.323, 104.66, 179]
  MoveL 1912 to (224.46, 47.08, -16.48) mm, rotated rx 180 ry 0 rz -49.48 deg; joints [-4.653, -87.867, 145.823, -197.22, 6.343, 104.611, 179]
  MoveL 1913 to (224.69, 47.18, -16.48) mm, rotated rx -180 ry 0 rz -49.46 deg; joints [-4.654, -87.875, 145.847, -197.151, 6.372, 104.542, 179]
  MoveL 1914 to (224.92, 47.31, -16.48) mm, rotated rx 180 ry 0 rz -49.44 deg; joints [-4.655, -87.882, 145.874, -197.06, 6.411, 104.449, 179]
  MoveL 1915 to (225.07, 47.42, -16.47) mm, rotated rx 180 ry 0 rz -49.42 deg; joints [-4.656, -87.886, 145.895, -196.981, 6.444, 104.37, 179]
  MoveL 1916 to (225.23, 47.54, -16.47) mm, rotated rx -180 ry 0 rz -49.4 deg; joints [-4.657, -87.889, 145.917, -196.888, 6.484, 104.277, 179]
  MoveL 1917 to (225.39, 47.67, -16.47) mm, rotated rx -180 ry 0 rz -49.38 deg; joints [-4.658, -87.891, 145.942, -196.781, 6.53, 104.168, 179]
  MoveL 1918 to (225.55, 47.83, -16.48) mm, rotated rx -180 ry 0 rz -49.35 deg; joints [-4.659, -87.892, 145.97, -196.655, 6.585, 104.041, 179]
  MoveL 1919 to (225.66, 47.96, -16.47) mm, rotated rx -180 ry 0 rz -49.32 deg; joints [-4.659, -87.892, 145.992, -196.55, 6.632, 103.936, 179]
  MoveL 1920 to (225.77, 48.09, -16.47) mm, rotated rx -180 ry 0 rz -49.3 deg; joints [-4.66, -87.891, 146.013, -196.445, 6.679, 103.83, 179]
  MoveL 1921 to (225.86, 48.22, -16.48) mm, rotated rx 180 ry 0 rz -49.27 deg; joints [-4.661, -87.889, 146.034, -196.339, 6.727, 103.724, 179]
  MoveL 1922 to (225.94, 48.35, -16.48) mm, rotated rx -180 ry 0 rz -49.24 deg; joints [-4.662, -87.886, 146.055, -196.234, 6.776, 103.618, 179]
  MoveL 1923 to (226.07, 48.57, -16.47) mm, rotated rx 180 ry 0 rz -49.19 deg; joints [-4.663, -87.881, 146.089, -196.053, 6.86, 103.436, 179]
  MoveL 1924 to (226.17, 48.8, -16.47) mm, rotated rx -180 ry 0 rz -49.15 deg; joints [-4.664, -87.874, 146.122, -195.874, 6.946, 103.256, 179]
  MoveL 1925 to (226.25, 49.02, -16.48) mm, rotated rx -180 ry 0 rz -49.1 deg; joints [-4.665, -87.865, 146.154, -195.697, 7.034, 103.078, 179]
  MoveL 1926 to (226.31, 49.24, -16.47) mm, rotated rx 180 ry 0 rz -49.04 deg; joints [-4.666, -87.855, 146.185, -195.521, 7.123, 102.901, 179]
  MoveL 1927 to (226.36, 49.48, -16.47) mm, rotated rx -180 ry 0 rz -48.99 deg; joints [-4.667, -87.843, 146.218, -195.332, 7.221, 102.711, 179]
  MoveL 1928 to (226.39, 49.73, -16.48) mm, rotated rx -180 ry 0 rz -48.93 deg; joints [-4.668, -87.83, 146.25, -195.146, 7.32, 102.524, 179]
  MoveL 1929 to (226.4, 50.21, -16.47) mm, rotated rx 180 ry 0 rz -48.82 deg; joints [-4.67, -87.8, 146.312, -194.781, 7.522, 102.158, 179]
  MoveL 1930 to (226.4, 428.49, -16.48) mm, rotated rx -180 ry 0 rz -39.17 deg; joints [-4.906, -49.014, 151.017, -182.854, 60.435, 89.107, 179]
  MoveL 1931 to (226.4, 428.74, -16.48) mm, rotated rx 180 ry 0 rz -39.16 deg; joints [-4.906, -48.982, 151.014, -182.854, 60.478, 89.106, 179]
  MoveL 1932 to (226.38, 428.98, -16.48) mm, rotated rx -180 ry 0 rz -39.14 deg; joints [-4.906, -48.949, 151.01, -182.853, 60.522, 89.104, 179]
  MoveL 1933 to (226.35, 429.22, -16.48) mm, rotated rx -180 ry 0 rz -39.13 deg; joints [-4.907, -48.915, 151.005, -182.853, 60.568, 89.103, 179]
  MoveL 1934 to (226.29, 429.46, -16.48) mm, rotated rx -180 ry 0 rz -39.11 deg; joints [-4.907, -48.88, 150.999, -182.852, 60.616, 89.101, 179]
  MoveL 1935 to (226.22, 429.7, -16.47) mm, rotated rx 180 ry 0 rz -39.08 deg; joints [-4.907, -48.844, 150.991, -182.852, 60.666, 89.1, 179]
  MoveL 1936 to (226.12, 429.94, -16.48) mm, rotated rx -180 ry 0 rz -39.06 deg; joints [-4.907, -48.806, 150.983, -182.852, 60.718, 89.098, 179]
  MoveL 1937 to (226.04, 430.11, -16.48) mm, rotated rx -180 ry 0 rz -39.04 deg; joints [-4.907, -48.78, 150.976, -182.852, 60.755, 89.097, 179]
  MoveL 1938 to (225.94, 430.28, -16.48) mm, rotated rx -180 ry 0 rz -39.02 deg; joints [-4.907, -48.753, 150.969, -182.851, 60.794, 89.096, 179]
  MoveL 1939 to (225.86, 430.4, -16.48) mm, rotated rx -180 ry 0 rz -39.01 deg; joints [-4.907, -48.732, 150.963, -182.851, 60.824, 89.095, 179]
  MoveL 1940 to (225.77, 430.53, -16.48) mm, rotated rx -180 ry 0 rz -38.99 deg; joints [-4.907, -48.711, 150.957, -182.851, 60.854, 89.095, 179]
  MoveL 1941 to (225.67, 430.65, -16.48) mm, rotated rx -180 ry 0 rz -38.98 deg; joints [-4.907, -48.69, 150.95, -182.851, 60.886, 89.094, 179]
  MoveL 1942 to (225.57, 430.78, -16.48) mm, rotated rx -180 ry 0 rz -38.96 deg; joints [-4.906, -48.668, 150.942, -182.851, 60.919, 89.093, 179]
  MoveL 1943 to (225.42, 430.93, -16.48) mm, rotated rx -180 ry 0 rz -38.93 deg; joints [-4.906, -48.64, 150.932, -182.85, 60.96, 89.093, 179]
  MoveL 1944 to (225.27, 431.06, -16.47) mm, rotated rx 180 ry 0 rz -38.91 deg; joints [-4.906, -48.615, 150.923, -182.85, 60.998, 89.092, 179]
  MoveL 1945 to (225.12, 431.17, -16.48) mm, rotated rx -180 ry 0 rz -38.89 deg; joints [-4.906, -48.592, 150.913, -182.85, 61.033, 89.092, 179]
  MoveL 1946 to (224.98, 431.28, -16.48) mm, rotated rx -180 ry 0 rz -38.87 deg; joints [-4.906, -48.571, 150.904, -182.85, 61.066, 89.091, 179]
  MoveL 1947 to (224.74, 431.42, -16.48) mm, rotated rx 180 ry 0 rz -38.84 deg; joints [-4.905, -48.54, 150.889, -182.85, 61.115, 89.091, 179]
  MoveL 1948 to (224.5, 431.54, -16.48) mm, rotated rx 180 ry 0 rz -38.8 deg; joints [-4.905, -48.512, 150.875, -182.85, 61.16, 89.09, 179]
  MoveL 1949 to (224.25, 431.63, -16.48) mm, rotated rx -180 ry 0 rz -38.77 deg; joints [-4.904, -48.488, 150.86, -182.849, 61.201, 89.09, 179]
  MoveL 1950 to (224.01, 431.7, -16.48) mm, rotated rx 180 ry 0 rz -38.75 deg; joints [-4.904, -48.466, 150.847, -182.849, 61.238, 89.09, 179]
  MoveL 1951 to (223.77, 431.76, -16.47) mm, rotated rx 180 ry 0 rz -38.72 deg; joints [-4.903, -48.447, 150.833, -182.849, 61.271, 89.09, 179]
  MoveL 1952 to (223.53, 431.79, -16.48) mm, rotated rx -180 ry 0 rz -38.69 deg; joints [-4.903, -48.431, 150.82, -182.849, 61.301, 89.09, 179]
  MoveL 1953 to (223.29, 431.8, -16.47) mm, rotated rx 180 ry 0 rz -38.66 deg; joints [-4.902, -48.417, 150.807, -182.849, 61.328, 89.091, 179]
  MoveL 1954 to (223.05, 431.8, -16.47) mm, rotated rx 180 ry 0 rz -38.64 deg; joints [-4.902, -48.404, 150.794, -182.849, 61.353, 89.091, 179]
  MoveL 1955 to (-164.9, 431.8, -16.48) mm, rotated rx 180 ry 0 rz 9.58 deg; joints [-4.404, -32.058, 134.415, -182.795, 89.641, 89.31, 159.098]
  MoveL 1956 to (-194.97, 431.99, -17.52) mm, rotated rx 180 ry 0 rz 12.97 deg; joints [-4.464, -31.102, 133.986, -182.853, 90.167, 89.271, 155.709]
  MoveL 1957 to (-195.47, 431.99, -17.52) mm, rotated rx 180 ry 0 rz 13.03 deg; joints [-4.464, -31.086, 133.979, -182.853, 90.176, 89.271, 155.654]
